gfCNCPoint1[22811] = {X 129.1532, Y 40.1052, Z -2.1667, A 0.000, B 0.000, C 0.000 }
gfCNCPoint1[22812] = {X 131.4548, Y 40.7854, Z -2.1667, A 0.000, B 0.000, C 0.000 }
gfCNCPoint1[22813] = {X 131.9017, Y 39.5320, Z -2.1667, A 0.000, B 0.000, C 0.000 }
gfCNCPoint1[22814] = {X 132.4836, Y 38.3354, Z -2.1667, A 0.000, B 0.000, C 0.000 }
gfCNCPoint1[22815] = {X 132.4836, Y 29.5202, Z -2.1667, A 0.000, B 0.000, C 0.000 }
gfCNCPoint1[22816] = {X 131.3523, Y 29.3993, Z -2.1667, A 0.000, B 0.000, C 0.000 }
gfCNCPoint1[22817] = {X 130.2373, Y 29.1724, Z -2.1667, A 0.000, B 0.000, C 0.000 }
gfCNCPoint1[22818] = {X 129.1487, Y 28.8417, Z -2.1667, A 0.000, B 0.000, C 0.000 }
gfCNCPoint1[22819] = {X 128.0242, Y 28.3763, Z -2.1667, A 0.000, B 0.000, C 0.000 }
gfCNCPoint1[22820] = {X 126.9523, Y 27.8001, Z -2.1667, A 0.000, B 0.000, C 0.000 }
gfCNCPoint1[22821] = {X 125.9438, Y 27.1189, Z -2.1667, A 0.000, B 0.000, C 0.000 }
gfCNCPoint1[22822] = {X 125.9432, Y 38.9884, Z -2.1667, A 0.000, B 0.000, C 0.000 }
gfCNCPoint1[22823] = {X 126.4735, Y 39.9279, Z -2.1667, A 0.000, B 0.000, C 0.000 }
gfCNCPoint1[22824] = {X 126.8960, Y 40.9205, Z -2.1667, A 0.000, B 0.000, C 0.000 }
gfCNCPoint1[22825] = {X 127.2098, Y 41.9730, Z -2.1667, A 0.000, B 0.000, C 0.000 }
gfCNCPoint1[22826] = {X 127.4025, Y 43.0542, Z -2.1667, A 0.000, B 0.000, C 0.000 }
gfCNCPoint1[22827] = {X 127.4714, Y 44.1502, Z -2.1667, A 0.000, B 0.000, C 0.000 }
gfCNCPoint1[22828] = {X 127.4716, Y 45.0000, Z -2.1667, A 0.000, B 0.000, C 0.000 }
gfCNCPoint1[22829] = {X 127.4070, Y 46.1159, Z -2.1667, A 0.000, B 0.000, C 0.000 }
gfCNCPoint1[22830] = {X 127.2143, Y 47.2168, Z -2.1667, A 0.000, B 0.000, C 0.000 }
gfCNCPoint1[22831] = {X 126.8960, Y 48.2883, Z -2.1667, A 0.000, B 0.000, C 0.000 }
gfCNCPoint1[22832] = {X 126.2883, Y 49.6376, Z -2.1667, A 0.000, B 0.000, C 0.000 }
gfCNCPoint1[22833] = {X 125.4821, Y 50.8786, Z -2.1667, A 0.000, B 0.000, C 0.000 }
gfCNCPoint1[22834] = {X 124.4962, Y 51.9821, Z -2.1667, A 0.000, B 0.000, C 0.000 }
gfCNCPoint1[22835] = {X 123.3536, Y 52.9225, Z -2.1667, A 0.000, B 0.000, C 0.000 }
gfCNCPoint1[22836] = {X 122.0810, Y 53.6778, Z -2.1667, A 0.000, B 0.000, C 0.000 }
gfCNCPoint1[22837] = {X 120.7081, Y 54.2302, Z -2.1667, A 0.000, B 0.000, C 0.000 }
gfCNCPoint1[22838] = {X 119.2671, Y 54.5669, Z -2.1667, A 0.000, B 0.000, C 0.000 }
gfCNCPoint1[22839] = {X 117.7916, Y 54.6800, Z -2.1667, A 0.000, B 0.000, C 0.000 }
gfCNCPoint1[22840] = {X 111.9185, Y 54.6800, Z -2.1667, A 0.000, B 0.000, C 0.000 }
gfCNCPoint1[22841] = {X 110.6386, Y 54.5950, Z -2.1667, A 0.000, B 0.000, C 0.000 }
gfCNCPoint1[22842] = {X 109.3812, Y 54.3415, Z -2.1667, A 0.000, B 0.000, C 0.000 }
gfCNCPoint1[22843] = {X 108.1683, Y 53.9240, Z -2.1667, A 0.000, B 0.000, C 0.000 }
gfCNCPoint1[22844] = {X 107.0213, Y 53.3498, Z -2.1667, A 0.000, B 0.000, C 0.000 }
gfCNCPoint1[22845] = {X 106.6480, Y 53.5578, Z -2.1667, A 0.000, B 0.000, C 0.000 }
gfCNCPoint1[22846] = {X 106.2658, Y 53.7492, Z -2.1667, A 0.000, B 0.000, C 0.000 }
gfCNCPoint1[22847] = {X 105.0149, Y 54.2382, Z -2.1667, A 0.000, B 0.000, C 0.000 }
gfCNCPoint1[22848] = {X 103.7084, Y 54.5495, Z -2.1667, A 0.000, B 0.000, C 0.000 }
gfCNCPoint1[22849] = {X 102.3713, Y 54.6768, Z -2.1667, A 0.000, B 0.000, C 0.000 }
gfCNCPoint1[22850] = {X 101.0295, Y 54.6179, Z -2.1667, A 0.000, B 0.000, C 0.000 }
gfCNCPoint1[22851] = {X 99.7088, Y 54.3738, Z -2.1667, A 0.000, B 0.000, C 0.000 }
gfCNCPoint1[22852] = {X 98.4345, Y 53.9493, Z -2.1667, A 0.000, B 0.000, C 0.000 }
gfCNCPoint1[22853] = {X 97.2313, Y 53.3524, Z -2.1667, A 0.000, B 0.000, C 0.000 }
gfCNCPoint1[22854] = {X 96.0852, Y 53.9255, Z -2.1667, A 0.000, B 0.000, C 0.000 }
gfCNCPoint1[22855] = {X 94.8734, Y 54.3422, Z -2.1667, A 0.000, B 0.000, C 0.000 }
gfCNCPoint1[22856] = {X 93.6172, Y 54.5952, Z -2.1667, A 0.000, B 0.000, C 0.000 }
gfCNCPoint1[22857] = {X 92.3385, Y 54.6800, Z -2.1667, A 0.000, B 0.000, C 0.000 }
gfCNCPoint1[22858] = {X 85.8951, Y 54.6800, Z -2.1667, A 0.000, B 0.000, C 0.000 }
gfCNCPoint1[22859] = {X 84.6159, Y 54.5951, Z -2.1667, A 0.000, B 0.000, C 0.000 }
gfCNCPoint1[22860] = {X 83.3592, Y 54.3419, Z -2.1667, A 0.000, B 0.000, C 0.000 }
gfCNCPoint1[22861] = {X 82.1469, Y 53.9249, Z -2.1667, A 0.000, B 0.000, C 0.000 }
gfCNCPoint1[22862] = {X 81.0644, Y 55.1572, Z -2.1667, A 0.000, B 0.000, C 0.000 }
gfCNCPoint1[22863] = {X 79.8495, Y 56.2591, Z -2.1667, A 0.000, B 0.000, C 0.000 }
gfCNCPoint1[22864] = {X 78.5178, Y 57.2166, Z -2.1667, A 0.000, B 0.000, C 0.000 }
gfCNCPoint1[22865] = {X 77.0863, Y 58.0174, Z -2.1667, A 0.000, B 0.000, C 0.000 }
gfCNCPoint1[22866] = {X 75.5734, Y 58.6511, Z -2.1667, A 0.000, B 0.000, C 0.000 }
gfCNCPoint1[22867] = {X 73.9986, Y 59.1096, Z -2.1667, A 0.000, B 0.000, C 0.000 }
gfCNCPoint1[22868] = {X 72.3820, Y 59.3871, Z -2.1667, A 0.000, B 0.000, C 0.000 }
gfCNCPoint1[22869] = {X 70.7445, Y 59.4800, Z -2.1667, A 0.000, B 0.000, C 0.000 }
gfCNCPoint1[22870] = {X 64.1851, Y 59.4800, Z -2.1667, A 0.000, B 0.000, C 0.000 }
gfCNCPoint1[22871] = {X 62.4203, Y 59.3720, Z -2.1667, A 0.000, B 0.000, C 0.000 }
gfCNCPoint1[22872] = {X 60.6818, Y 59.0498, Z -2.1667, A 0.000, B 0.000, C 0.000 }
gfCNCPoint1[22873] = {X 58.9955, Y 58.5181, Z -2.1667, A 0.000, B 0.000, C 0.000 }
gfCNCPoint1[22874] = {X 57.3866, Y 57.7848, Z -2.1667, A 0.000, B 0.000, C 0.000 }
gfCNCPoint1[22875] = {X 55.8790, Y 56.8608, Z -2.1667, A 0.000, B 0.000, C 0.000 }
gfCNCPoint1[22876] = {X 54.3715, Y 57.7848, Z -2.1667, A 0.000, B 0.000, C 0.000 }
gfCNCPoint1[22877] = {X 52.7626, Y 58.5181, Z -2.1667, A 0.000, B 0.000, C 0.000 }
gfCNCPoint1[22878] = {X 51.0763, Y 59.0498, Z -2.1667, A 0.000, B 0.000, C 0.000 }
gfCNCPoint1[22879] = {X 49.3378, Y 59.3720, Z -2.1667, A 0.000, B 0.000, C 0.000 }
gfCNCPoint1[22880] = {X 47.5729, Y 59.4800, Z -2.1667, A 0.000, B 0.000, C 0.000 }
gfCNCPoint1[22881] = {X 40.6393, Y 59.4800, Z -2.1667, A 0.000, B 0.000, C 0.000 }
gfCNCPoint1[22882] = {X 38.9795, Y 59.3845, Z -2.1667, A 0.000, B 0.000, C 0.000 }
gfCNCPoint1[22883] = {X 37.3415, Y 59.0995, Z -2.1667, A 0.000, B 0.000, C 0.000 }
gfCNCPoint1[22884] = {X 35.7470, Y 58.6285, Z -2.1667, A 0.000, B 0.000, C 0.000 }
gfCNCPoint1[22885] = {X 34.0331, Y 59.4863, Z -2.1667, A 0.000, B 0.000, C 0.000 }
gfCNCPoint1[22886] = {X 32.2408, Y 60.1653, Z -2.1667, A 0.000, B 0.000, C 0.000 }
gfCNCPoint1[22887] = {X 30.3888, Y 60.6585, Z -2.1667, A 0.000, B 0.000, C 0.000 }
gfCNCPoint1[22888] = {X 28.4962, Y 60.9608, Z -2.1667, A 0.000, B 0.000, C 0.000 }
gfCNCPoint1[22889] = {X 25.7981, Y 62.0563, Z -2.1667, A 0.000, B 0.000, C 0.000 }
gfCNCPoint1[22890] = {X 23.0321, Y 62.9667, Z -2.1667, A 0.000, B 0.000, C 0.000 }
gfCNCPoint1[22891] = {X 20.1653, Y 63.6947, Z -2.1667, A 0.000, B 0.000, C 0.000 }
gfCNCPoint1[22892] = {X 17.2496, Y 64.1921, Z -2.1667, A 0.000, B 0.000, C 0.000 }
gfCNCPoint1[22893] = {X 14.3035, Y 64.4558, Z -2.1667, A 0.000, B 0.000, C 0.000 }
gfCNCPoint1[22894] = {X 14.3035, Y 85.6949, Z -2.1667, A 0.000, B 0.000, C 0.000 }
gfCNCPoint1[22895] = {X 112.5246, Y 85.6949, Z -2.1667, A 0.000, B 0.000, C 0.000 }
gfCNCPoint1[22896] = {X 113.6274, Y 84.5920, Z -2.1667, A 0.000, B 0.000, C 0.000 }
gfCNCPoint1[22897] = {X 114.8273, Y 83.5956, Z -2.1667, A 0.000, B 0.000, C 0.000 }
gfCNCPoint1[22898] = {X 116.1140, Y 82.7142, Z -2.1667, A 0.000, B 0.000, C 0.000 }
gfCNCPoint1[22899] = {X 117.4766, Y 81.9553, Z -2.1667, A 0.000, B 0.000, C 0.000 }
gfCNCPoint1[22900] = {X 111.0585, Y 69.0646, Z -2.1667, A 0.000, B 0.000, C 0.000 }
gfCNCPoint1[22901] = {X 109.0296, Y 68.9061, Z -2.1667, A 0.000, B 0.000, C 0.000 }
gfCNCPoint1[22902] = {X 107.0213, Y 68.5768, Z -2.1667, A 0.000, B 0.000, C 0.000 }
gfCNCPoint1[22903] = {X 105.0765, Y 68.8983, Z -2.1667, A 0.000, B 0.000, C 0.000 }
gfCNCPoint1[22904] = {X 103.1119, Y 69.0597, Z -2.1667, A 0.000, B 0.000, C 0.000 }
gfCNCPoint1[22905] = {X 101.1407, Y 69.0599, Z -2.1667, A 0.000, B 0.000, C 0.000 }
gfCNCPoint1[22906] = {X 99.1761, Y 68.8989, Z -2.1667, A 0.000, B 0.000, C 0.000 }
gfCNCPoint1[22907] = {X 97.2313, Y 68.5777, Z -2.1667, A 0.000, B 0.000, C 0.000 }
gfCNCPoint1[22908] = {X 95.6131, Y 68.8563, Z -2.1667, A 0.000, B 0.000, C 0.000 }
gfCNCPoint1[22909] = {X 93.9796, Y 69.0240, Z -2.1667, A 0.000, B 0.000, C 0.000 }
gfCNCPoint1[22910] = {X 92.3385, Y 69.0800, Z -2.1667, A 0.000, B 0.000, C 0.000 }
gfCNCPoint1[22911] = {X 86.6884, Y 69.0800, Z -2.1667, A 0.000, B 0.000, C 0.000 }
gfCNCPoint1[22912] = {X 84.7317, Y 70.2668, Z -2.1667, A 0.000, B 0.000, C 0.000 }
gfCNCPoint1[22913] = {X 82.6873, Y 71.2949, Z -2.1667, A 0.000, B 0.000, C 0.000 }
gfCNCPoint1[22914] = {X 107.2717, Y 71.2949, Z -2.1667, A 0.000, B 0.000, C 0.000 }
gfCNCPoint1[22915] = {X 109.1259, Y 70.1132, Z -2.1667, A 0.000, B 0.000, C 0.000 }
gfCNCPoint1[22916] = {X 111.0585, Y 69.0646, Z -2.1667, A 0.000, B 0.000, C 0.000 }
gfCNCPoint1[22917] = {X 112.1282, Y 71.2131, Z -2.1667, A 0.000, B 0.000, C 0.000 }
gfCNCPoint1[22918] = {X 113.1274, Y 70.7392, Z -2.1667, A 0.000, B 0.000, C 0.000 }
gfCNCPoint1[22919] = {X 114.1439, Y 70.3040, Z -2.1667, A 0.000, B 0.000, C 0.000 }
gfCNCPoint1[22920] = {X 117.4441, Y 66.6800, Z -2.1667, A 0.000, B 0.000, C 0.000 }
gfCNCPoint1[22921] = {X 111.9185, Y 66.6800, Z -2.1667, A 0.000, B 0.000, C 0.000 }
gfCNCPoint1[22922] = {X 111.5313, Y 66.6765, Z -2.1667, A 0.000, B 0.000, C 0.000 }
gfCNCPoint1[22923] = {X 111.1442, Y 66.6662, Z -2.1667, A 0.000, B 0.000, C 0.000 }
gfCNCPoint1[22924] = {X 109.0696, Y 66.4920, Z -2.1667, A 0.000, B 0.000, C 0.000 }
gfCNCPoint1[22925] = {X 107.0213, Y 66.1197, Z -2.1667, A 0.000, B 0.000, C 0.000 }
gfCNCPoint1[22926] = {X 105.0796, Y 66.4776, Z -2.1667, A 0.000, B 0.000, C 0.000 }
gfCNCPoint1[22927] = {X 103.1135, Y 66.6574, Z -2.1667, A 0.000, B 0.000, C 0.000 }
gfCNCPoint1[22928] = {X 101.1392, Y 66.6576, Z -2.1667, A 0.000, B 0.000, C 0.000 }
gfCNCPoint1[22929] = {X 99.1730, Y 66.4782, Z -2.1667, A 0.000, B 0.000, C 0.000 }
gfCNCPoint1[22930] = {X 97.2313, Y 66.1207, Z -2.1667, A 0.000, B 0.000, C 0.000 }
gfCNCPoint1[22931] = {X 95.6161, Y 66.4308, Z -2.1667, A 0.000, B 0.000, C 0.000 }
gfCNCPoint1[22932] = {X 93.9821, Y 66.6176, Z -2.1667, A 0.000, B 0.000, C 0.000 }
gfCNCPoint1[22933] = {X 92.3385, Y 66.6800, Z -2.1667, A 0.000, B 0.000, C 0.000 }
gfCNCPoint1[22934] = {X 85.9487, Y 66.6800, Z -2.1667, A 0.000, B 0.000, C 0.000 }
gfCNCPoint1[22935] = {X 83.8781, Y 67.9935, Z -2.1667, A 0.000, B 0.000, C 0.000 }
gfCNCPoint1[22936] = {X 81.6948, Y 69.1097, Z -2.1667, A 0.000, B 0.000, C 0.000 }
gfCNCPoint1[22937] = {X 79.6018, Y 69.9547, Z -2.1667, A 0.000, B 0.000, C 0.000 }
gfCNCPoint1[22938] = {X 77.4444, Y 70.6184, Z -2.1667, A 0.000, B 0.000, C 0.000 }
gfCNCPoint1[22939] = {X 75.2383, Y 71.0959, Z -2.1667, A 0.000, B 0.000, C 0.000 }
gfCNCPoint1[22940] = {X 72.9996, Y 71.3838, Z -2.1667, A 0.000, B 0.000, C 0.000 }
gfCNCPoint1[22941] = {X 70.7445, Y 71.4800, Z -2.1667, A 0.000, B 0.000, C 0.000 }
gfCNCPoint1[22942] = {X 64.1851, Y 71.4800, Z -2.1667, A 0.000, B 0.000, C 0.000 }
gfCNCPoint1[22943] = {X 62.0752, Y 71.3958, Z -2.1667, A 0.000, B 0.000, C 0.000 }
gfCNCPoint1[22944] = {X 59.9787, Y 71.1438, Z -2.1667, A 0.000, B 0.000, C 0.000 }
gfCNCPoint1[22945] = {X 57.9089, Y 70.7255, Z -2.1667, A 0.000, B 0.000, C 0.000 }
gfCNCPoint1[22946] = {X 55.8790, Y 70.1436, Z -2.1667, A 0.000, B 0.000, C 0.000 }
gfCNCPoint1[22947] = {X 53.8492, Y 70.7255, Z -2.1667, A 0.000, B 0.000, C 0.000 }
gfCNCPoint1[22948] = {X 51.7794, Y 71.1438, Z -2.1667, A 0.000, B 0.000, C 0.000 }
gfCNCPoint1[22949] = {X 49.6829, Y 71.3958, Z -2.1667, A 0.000, B 0.000, C 0.000 }
gfCNCPoint1[22950] = {X 47.5729, Y 71.4800, Z -2.1667, A 0.000, B 0.000, C 0.000 }
gfCNCPoint1[22951] = {X 40.6393, Y 71.4800, Z -2.1667, A 0.000, B 0.000, C 0.000 }
gfCNCPoint1[22952] = {X 38.8042, Y 71.4163, Z -2.1667, A 0.000, B 0.000, C 0.000 }
gfCNCPoint1[22953] = {X 36.9779, Y 71.2256, Z -2.1667, A 0.000, B 0.000, C 0.000 }
gfCNCPoint1[22954] = {X 34.3998, Y 72.0339, Z -2.1667, A 0.000, B 0.000, C 0.000 }
gfCNCPoint1[22955] = {X 31.7610, Y 72.6132, Z -2.1667, A 0.000, B 0.000, C 0.000 }
gfCNCPoint1[22956] = {X 30.3294, Y 73.1742, Z -2.1667, A 0.000, B 0.000, C 0.000 }
gfCNCPoint1[22957] = {X 28.8828, Y 73.6949, Z -2.1667, A 0.000, B 0.000, C 0.000 }
gfCNCPoint1[22958] = {X 108.0339, Y 73.6949, Z -2.1667, A 0.000, B 0.000, C 0.000 }
gfCNCPoint1[22959] = {X 110.0295, Y 72.3690, Z -2.1667, A 0.000, B 0.000, C 0.000 }
gfCNCPoint1[22960] = {X 112.1282, Y 71.2131, Z -2.1667, A 0.000, B 0.000, C 0.000 }
gfCNCPoint1[22961] = {X 113.1979, Y 73.3615, Z -2.1667, A 0.000, B 0.000, C 0.000 }
gfCNCPoint1[22962] = {X 114.3580, Y 72.8185, Z -2.1667, A 0.000, B 0.000, C 0.000 }
gfCNCPoint1[22963] = {X 115.5430, Y 72.3323, Z -2.1667, A 0.000, B 0.000, C 0.000 }
gfCNCPoint1[22964] = {X 123.7288, Y 63.3431, Z -2.1667, A 0.000, B 0.000, C 0.000 }
gfCNCPoint1[22965] = {X 121.7860, Y 63.8617, Z -2.1667, A 0.000, B 0.000, C 0.000 }
gfCNCPoint1[22966] = {X 119.7997, Y 64.1751, Z -2.1667, A 0.000, B 0.000, C 0.000 }
gfCNCPoint1[22967] = {X 117.7916, Y 64.2800, Z -2.1667, A 0.000, B 0.000, C 0.000 }
gfCNCPoint1[22968] = {X 111.9185, Y 64.2800, Z -2.1667, A 0.000, B 0.000, C 0.000 }
gfCNCPoint1[22969] = {X 110.2700, Y 64.2094, Z -2.1667, A 0.000, B 0.000, C 0.000 }
gfCNCPoint1[22970] = {X 108.6336, Y 63.9981, Z -2.1667, A 0.000, B 0.000, C 0.000 }
gfCNCPoint1[22971] = {X 107.0213, Y 63.6477, Z -2.1667, A 0.000, B 0.000, C 0.000 }
gfCNCPoint1[22972] = {X 105.0841, Y 64.0514, Z -2.1667, A 0.000, B 0.000, C 0.000 }
gfCNCPoint1[22973] = {X 103.1158, Y 64.2545, Z -2.1667, A 0.000, B 0.000, C 0.000 }
gfCNCPoint1[22974] = {X 101.1370, Y 64.2547, Z -2.1667, A 0.000, B 0.000, C 0.000 }
gfCNCPoint1[22975] = {X 99.1686, Y 64.0521, Z -2.1667, A 0.000, B 0.000, C 0.000 }
gfCNCPoint1[22976] = {X 97.2313, Y 63.6488, Z -2.1667, A 0.000, B 0.000, C 0.000 }
gfCNCPoint1[22977] = {X 95.6204, Y 63.9986, Z -2.1667, A 0.000, B 0.000, C 0.000 }
gfCNCPoint1[22978] = {X 93.9855, Y 64.2095, Z -2.1667, A 0.000, B 0.000, C 0.000 }
gfCNCPoint1[22979] = {X 92.3385, Y 64.2800, Z -2.1667, A 0.000, B 0.000, C 0.000 }
gfCNCPoint1[22980] = {X 85.8951, Y 64.2800, Z -2.1667, A 0.000, B 0.000, C 0.000 }
gfCNCPoint1[22981] = {X 85.5417, Y 64.2768, Z -2.1667, A 0.000, B 0.000, C 0.000 }
gfCNCPoint1[22982] = {X 85.1884, Y 64.2670, Z -2.1667, A 0.000, B 0.000, C 0.000 }
gfCNCPoint1[22983] = {X 83.3593, Y 65.5113, Z -2.1667, A 0.000, B 0.000, C 0.000 }
gfCNCPoint1[22984] = {X 81.4238, Y 66.5824, Z -2.1667, A 0.000, B 0.000, C 0.000 }
gfCNCPoint1[22985] = {X 79.3981, Y 67.4713, Z -2.1667, A 0.000, B 0.000, C 0.000 }
gfCNCPoint1[22986] = {X 77.2994, Y 68.1706, Z -2.1667, A 0.000, B 0.000, C 0.000 }
gfCNCPoint1[22987] = {X 75.1454, Y 68.6744, Z -2.1667, A 0.000, B 0.000, C 0.000 }
gfCNCPoint1[22988] = {X 72.9543, Y 68.9784, Z -2.1667, A 0.000, B 0.000, C 0.000 }
gfCNCPoint1[22989] = {X 70.7445, Y 69.0800, Z -2.1667, A 0.000, B 0.000, C 0.000 }
gfCNCPoint1[22990] = {X 64.1851, Y 69.0800, Z -2.1667, A 0.000, B 0.000, C 0.000 }
gfCNCPoint1[22991] = {X 62.0678, Y 68.9867, Z -2.1667, A 0.000, B 0.000, C 0.000 }
gfCNCPoint1[22992] = {X 59.9669, Y 68.7076, Z -2.1667, A 0.000, B 0.000, C 0.000 }
gfCNCPoint1[22993] = {X 57.8986, Y 68.2449, Z -2.1667, A 0.000, B 0.000, C 0.000 }
gfCNCPoint1[22994] = {X 55.8790, Y 67.6021, Z -2.1667, A 0.000, B 0.000, C 0.000 }
gfCNCPoint1[22995] = {X 53.8595, Y 68.2449, Z -2.1667, A 0.000, B 0.000, C 0.000 }
gfCNCPoint1[22996] = {X 51.7912, Y 68.7076, Z -2.1667, A 0.000, B 0.000, C 0.000 }
gfCNCPoint1[22997] = {X 49.6903, Y 68.9867, Z -2.1667, A 0.000, B 0.000, C 0.000 }
gfCNCPoint1[22998] = {X 47.5729, Y 69.0800, Z -2.1667, A 0.000, B 0.000, C 0.000 }
gfCNCPoint1[22999] = {X 40.6393, Y 69.0800, Z -2.1667, A 0.000, B 0.000, C 0.000 }
gfCNCPoint1[23000] = {X 38.6738, Y 68.9996, Z -2.1667, A 0.000, B 0.000, C 0.000 }
gfCNCPoint1[23001] = {X 36.7214, Y 68.7591, Z -2.1667, A 0.000, B 0.000, C 0.000 }
gfCNCPoint1[23002] = {X 34.8828, Y 69.3981, Z -2.1667, A 0.000, B 0.000, C 0.000 }
gfCNCPoint1[23003] = {X 33.0048, Y 69.9097, Z -2.1667, A 0.000, B 0.000, C 0.000 }
gfCNCPoint1[23004] = {X 31.0962, Y 70.2916, Z -2.1667, A 0.000, B 0.000, C 0.000 }
gfCNCPoint1[23005] = {X 29.6075, Y 70.8814, Z -2.1667, A 0.000, B 0.000, C 0.000 }
gfCNCPoint1[23006] = {X 28.1016, Y 71.4256, Z -2.1667, A 0.000, B 0.000, C 0.000 }
gfCNCPoint1[23007] = {X 26.9268, Y 71.8147, Z -2.1667, A 0.000, B 0.000, C 0.000 }
gfCNCPoint1[23008] = {X 25.7433, Y 72.1759, Z -2.1667, A 0.000, B 0.000, C 0.000 }
gfCNCPoint1[23009] = {X 24.8260, Y 72.4376, Z -2.1667, A 0.000, B 0.000, C 0.000 }
gfCNCPoint1[23010] = {X 23.9035, Y 72.6805, Z -2.1667, A 0.000, B 0.000, C 0.000 }
gfCNCPoint1[23011] = {X 23.9035, Y 76.0949, Z -2.1667, A 0.000, B 0.000, C 0.000 }
gfCNCPoint1[23012] = {X 108.8319, Y 76.0949, Z -2.1667, A 0.000, B 0.000, C 0.000 }
gfCNCPoint1[23013] = {X 110.2270, Y 75.0898, Z -2.1667, A 0.000, B 0.000, C 0.000 }
gfCNCPoint1[23014] = {X 111.6843, Y 74.1774, Z -2.1667, A 0.000, B 0.000, C 0.000 }
gfCNCPoint1[23015] = {X 113.1979, Y 73.3615, Z -2.1667, A 0.000, B 0.000, C 0.000 }
gfCNCPoint1[23016] = {X 114.2675, Y 75.5099, Z -2.1667, A 0.000, B 0.000, C 0.000 }
gfCNCPoint1[23017] = {X 115.5786, Y 74.9055, Z -2.1667, A 0.000, B 0.000, C 0.000 }
gfCNCPoint1[23018] = {X 116.9235, Y 74.3808, Z -2.1667, A 0.000, B 0.000, C 0.000 }
gfCNCPoint1[23019] = {X 130.4117, Y 59.5689, Z -2.1667, A 0.000, B 0.000, C 0.000 }
gfCNCPoint1[23020] = {X 129.5280, Y 58.7534, Z -2.1667, A 0.000, B 0.000, C 0.000 }
gfCNCPoint1[23021] = {X 128.6970, Y 57.8844, Z -2.1667, A 0.000, B 0.000, C 0.000 }
gfCNCPoint1[23022] = {X 127.3931, Y 58.8832, Z -2.1667, A 0.000, B 0.000, C 0.000 }
gfCNCPoint1[23023] = {X 125.9984, Y 59.7507, Z -2.1667, A 0.000, B 0.000, C 0.000 }
gfCNCPoint1[23024] = {X 124.5259, Y 60.4785, Z -2.1667, A 0.000, B 0.000, C 0.000 }
gfCNCPoint1[23025] = {X 122.9897, Y 61.0597, Z -2.1667, A 0.000, B 0.000, C 0.000 }
gfCNCPoint1[23026] = {X 121.2887, Y 61.5138, Z -2.1667, A 0.000, B 0.000, C 0.000 }
gfCNCPoint1[23027] = {X 119.5497, Y 61.7882, Z -2.1667, A 0.000, B 0.000, C 0.000 }
gfCNCPoint1[23028] = {X 117.7916, Y 61.8800, Z -2.1667, A 0.000, B 0.000, C 0.000 }
gfCNCPoint1[23029] = {X 111.9185, Y 61.8800, Z -2.1667, A 0.000, B 0.000, C 0.000 }
gfCNCPoint1[23030] = {X 110.2649, Y 61.7988, Z -2.1667, A 0.000, B 0.000, C 0.000 }
gfCNCPoint1[23031] = {X 108.6273, Y 61.5560, Z -2.1667, A 0.000, B 0.000, C 0.000 }
gfCNCPoint1[23032] = {X 107.0213, Y 61.1540, Z -2.1667, A 0.000, B 0.000, C 0.000 }
gfCNCPoint1[23033] = {X 105.0907, Y 61.6173, Z -2.1667, A 0.000, B 0.000, C 0.000 }
gfCNCPoint1[23034] = {X 103.1191, Y 61.8506, Z -2.1667, A 0.000, B 0.000, C 0.000 }
gfCNCPoint1[23035] = {X 101.1337, Y 61.8509, Z -2.1667, A 0.000, B 0.000, C 0.000 }
gfCNCPoint1[23036] = {X 99.1620, Y 61.6181, Z -2.1667, A 0.000, B 0.000, C 0.000 }
gfCNCPoint1[23037] = {X 97.2313, Y 61.1553, Z -2.1667, A 0.000, B 0.000, C 0.000 }
gfCNCPoint1[23038] = {X 95.6267, Y 61.5566, Z -2.1667, A 0.000, B 0.000, C 0.000 }
gfCNCPoint1[23039] = {X 93.9906, Y 61.7990, Z -2.1667, A 0.000, B 0.000, C 0.000 }
gfCNCPoint1[23040] = {X 92.3385, Y 61.8800, Z -2.1667, A 0.000, B 0.000, C 0.000 }
gfCNCPoint1[23041] = {X 85.8951, Y 61.8800, Z -2.1667, A 0.000, B 0.000, C 0.000 }
gfCNCPoint1[23042] = {X 85.1609, Y 61.8640, Z -2.1667, A 0.000, B 0.000, C 0.000 }
gfCNCPoint1[23043] = {X 84.4280, Y 61.8161, Z -2.1667, A 0.000, B 0.000, C 0.000 }
gfCNCPoint1[23044] = {X 82.7246, Y 63.0692, Z -2.1667, A 0.000, B 0.000, C 0.000 }
gfCNCPoint1[23045] = {X 80.9073, Y 64.1504, Z -2.1667, A 0.000, B 0.000, C 0.000 }
gfCNCPoint1[23046] = {X 78.9932, Y 65.0494, Z -2.1667, A 0.000, B 0.000, C 0.000 }
gfCNCPoint1[23047] = {X 77.0007, Y 65.7577, Z -2.1667, A 0.000, B 0.000, C 0.000 }
gfCNCPoint1[23048] = {X 74.9487, Y 66.2685, Z -2.1667, A 0.000, B 0.000, C 0.000 }
gfCNCPoint1[23049] = {X 72.8566, Y 66.5769, Z -2.1667, A 0.000, B 0.000, C 0.000 }
gfCNCPoint1[23050] = {X 70.7445, Y 66.6800, Z -2.1667, A 0.000, B 0.000, C 0.000 }
gfCNCPoint1[23051] = {X 64.1851, Y 66.6800, Z -2.1667, A 0.000, B 0.000, C 0.000 }
gfCNCPoint1[23052] = {X 62.0576, Y 66.5753, Z -2.1667, A 0.000, B 0.000, C 0.000 }
gfCNCPoint1[23053] = {X 59.9505, Y 66.2624, Z -2.1667, A 0.000, B 0.000, C 0.000 }
gfCNCPoint1[23054] = {X 57.8844, Y 65.7442, Z -2.1667, A 0.000, B 0.000, C 0.000 }
gfCNCPoint1[23055] = {X 55.8790, Y 65.0258, Z -2.1667, A 0.000, B 0.000, C 0.000 }
gfCNCPoint1[23056] = {X 53.8737, Y 65.7442, Z -2.1667, A 0.000, B 0.000, C 0.000 }
gfCNCPoint1[23057] = {X 51.8075, Y 66.2624, Z -2.1667, A 0.000, B 0.000, C 0.000 }
gfCNCPoint1[23058] = {X 49.7005, Y 66.5753, Z -2.1667, A 0.000, B 0.000, C 0.000 }
gfCNCPoint1[23059] = {X 47.5729, Y 66.6800, Z -2.1667, A 0.000, B 0.000, C 0.000 }
gfCNCPoint1[23060] = {X 40.6393, Y 66.6800, Z -2.1667, A 0.000, B 0.000, C 0.000 }
gfCNCPoint1[23061] = {X 38.5440, Y 66.5785, Z -2.1667, A 0.000, B 0.000, C 0.000 }
gfCNCPoint1[23062] = {X 36.4684, Y 66.2750, Z -2.1667, A 0.000, B 0.000, C 0.000 }
gfCNCPoint1[23063] = {X 34.5052, Y 67.0002, Z -2.1667, A 0.000, B 0.000, C 0.000 }
gfCNCPoint1[23064] = {X 32.4901, Y 67.5653, Z -2.1667, A 0.000, B 0.000, C 0.000 }
gfCNCPoint1[23065] = {X 30.4361, Y 67.9665, Z -2.1667, A 0.000, B 0.000, C 0.000 }
gfCNCPoint1[23066] = {X 27.7779, Y 68.9963, Z -2.1667, A 0.000, B 0.000, C 0.000 }
gfCNCPoint1[23067] = {X 25.0655, Y 69.8736, Z -2.1667, A 0.000, B 0.000, C 0.000 }
gfCNCPoint1[23068] = {X 23.2938, Y 70.3591, Z -2.1667, A 0.000, B 0.000, C 0.000 }
gfCNCPoint1[23069] = {X 21.5035, Y 70.7708, Z -2.1667, A 0.000, B 0.000, C 0.000 }
gfCNCPoint1[23070] = {X 21.5035, Y 78.4949, Z -2.1667, A 0.000, B 0.000, C 0.000 }
gfCNCPoint1[23071] = {X 109.6715, Y 78.4949, Z -2.1667, A 0.000, B 0.000, C 0.000 }
gfCNCPoint1[23072] = {X 111.1263, Y 77.3843, Z -2.1667, A 0.000, B 0.000, C 0.000 }
gfCNCPoint1[23073] = {X 112.6613, Y 76.3874, Z -2.1667, A 0.000, B 0.000, C 0.000 }
gfCNCPoint1[23074] = {X 114.2675, Y 75.5099, Z -2.1667, A 0.000, B 0.000, C 0.000 }
gfCNCPoint1[23075] = {X 115.3372, Y 77.6584, Z -2.1667, A 0.000, B 0.000, C 0.000 }
gfCNCPoint1[23076] = {X 116.7878, Y 77.0015, Z -2.1667, A 0.000, B 0.000, C 0.000 }
gfCNCPoint1[23077] = {X 118.2826, Y 76.4529, Z -2.1667, A 0.000, B 0.000, C 0.000 }
gfCNCPoint1[23078] = {X 133.9639, Y 59.2326, Z -2.1667, A 0.000, B 0.000, C 0.000 }
gfCNCPoint1[23079] = {X 132.7159, Y 58.3550, Z -2.1667, A 0.000, B 0.000, C 0.000 }
gfCNCPoint1[23080] = {X 131.5522, Y 57.3683, Z -2.1667, A 0.000, B 0.000, C 0.000 }
gfCNCPoint1[23081] = {X 130.4824, Y 56.2805, Z -2.1667, A 0.000, B 0.000, C 0.000 }
gfCNCPoint1[23082] = {X 129.6655, Y 55.2988, Z -2.1667, A 0.000, B 0.000, C 0.000 }
gfCNCPoint1[23083] = {X 128.9251, Y 54.2582, Z -2.1667, A 0.000, B 0.000, C 0.000 }
gfCNCPoint1[23084] = {X 128.0750, Y 55.1942, Z -2.1667, A 0.000, B 0.000, C 0.000 }
gfCNCPoint1[23085] = {X 127.1464, Y 56.0525, Z -2.1667, A 0.000, B 0.000, C 0.000 }
gfCNCPoint1[23086] = {X 125.7915, Y 57.0695, Z -2.1667, A 0.000, B 0.000, C 0.000 }
gfCNCPoint1[23087] = {X 124.3270, Y 57.9212, Z -2.1667, A 0.000, B 0.000, C 0.000 }
gfCNCPoint1[23088] = {X 122.7731, Y 58.5961, Z -2.1667, A 0.000, B 0.000, C 0.000 }
gfCNCPoint1[23089] = {X 121.1510, Y 59.0849, Z -2.1667, A 0.000, B 0.000, C 0.000 }
gfCNCPoint1[23090] = {X 119.4828, Y 59.3809, Z -2.1667, A 0.000, B 0.000, C 0.000 }
gfCNCPoint1[23091] = {X 117.7916, Y 59.4800, Z -2.1667, A 0.000, B 0.000, C 0.000 }
gfCNCPoint1[23092] = {X 111.9185, Y 59.4800, Z -2.1667, A 0.000, B 0.000, C 0.000 }
gfCNCPoint1[23093] = {X 110.2569, Y 59.3844, Z -2.1667, A 0.000, B 0.000, C 0.000 }
gfCNCPoint1[23094] = {X 108.6173, Y 59.0987, Z -2.1667, A 0.000, B 0.000, C 0.000 }
gfCNCPoint1[23095] = {X 107.0213, Y 58.6267, Z -2.1667, A 0.000, B 0.000, C 0.000 }
gfCNCPoint1[23096] = {X 105.4260, Y 59.0985, Z -2.1667, A 0.000, B 0.000, C 0.000 }
gfCNCPoint1[23097] = {X 103.7872, Y 59.3842, Z -2.1667, A 0.000, B 0.000, C 0.000 }
gfCNCPoint1[23098] = {X 102.1264, Y 59.4800, Z -2.1667, A 0.000, B 0.000, C 0.000 }
gfCNCPoint1[23099] = {X 100.4656, Y 59.3847, Z -2.1667, A 0.000, B 0.000, C 0.000 }
gfCNCPoint1[23100] = {X 98.8267, Y 59.0996, Z -2.1667, A 0.000, B 0.000, C 0.000 }
gfCNCPoint1[23101] = {X 97.2313, Y 58.6283, Z -2.1667, A 0.000, B 0.000, C 0.000 }
gfCNCPoint1[23102] = {X 95.6367, Y 59.0994, Z -2.1667, A 0.000, B 0.000, C 0.000 }
gfCNCPoint1[23103] = {X 93.9986, Y 59.3845, Z -2.1667, A 0.000, B 0.000, C 0.000 }
gfCNCPoint1[23104] = {X 92.3385, Y 59.4800, Z -2.1667, A 0.000, B 0.000, C 0.000 }
gfCNCPoint1[23105] = {X 85.8951, Y 59.4800, Z -2.1667, A 0.000, B 0.000, C 0.000 }
gfCNCPoint1[23106] = {X 84.7780, Y 59.4368, Z -2.1667, A 0.000, B 0.000, C 0.000 }
gfCNCPoint1[23107] = {X 83.6677, Y 59.3077, Z -2.1667, A 0.000, B 0.000, C 0.000 }
gfCNCPoint1[23108] = {X 82.0978, Y 60.5827, Z -2.1667, A 0.000, B 0.000, C 0.000 }
gfCNCPoint1[23109] = {X 80.4031, Y 61.6862, Z -2.1667, A 0.000, B 0.000, C 0.000 }
gfCNCPoint1[23110] = {X 78.6021, Y 62.6061, Z -2.1667, A 0.000, B 0.000, C 0.000 }
gfCNCPoint1[23111] = {X 76.7146, Y 63.3324, Z -2.1667, A 0.000, B 0.000, C 0.000 }
gfCNCPoint1[23112] = {X 74.7614, Y 63.8569, Z -2.1667, A 0.000, B 0.000, C 0.000 }
gfCNCPoint1[23113] = {X 72.7640, Y 64.1739, Z -2.1667, A 0.000, B 0.000, C 0.000 }
gfCNCPoint1[23114] = {X 70.7445, Y 64.2800, Z -2.1667, A 0.000, B 0.000, C 0.000 }
gfCNCPoint1[23115] = {X 64.1851, Y 64.2800, Z -2.1667, A 0.000, B 0.000, C 0.000 }
gfCNCPoint1[23116] = {X 62.0428, Y 64.1606, Z -2.1667, A 0.000, B 0.000, C 0.000 }
gfCNCPoint1[23117] = {X 59.9269, Y 63.8039, Z -2.1667, A 0.000, B 0.000, C 0.000 }
gfCNCPoint1[23118] = {X 57.8638, Y 63.2143, Z -2.1667, A 0.000, B 0.000, C 0.000 }
gfCNCPoint1[23119] = {X 55.8790, Y 62.3991, Z -2.1667, A 0.000, B 0.000, C 0.000 }
gfCNCPoint1[23120] = {X 53.8942, Y 63.2143, Z -2.1667, A 0.000, B 0.000, C 0.000 }
gfCNCPoint1[23121] = {X 51.8311, Y 63.8039, Z -2.1667, A 0.000, B 0.000, C 0.000 }
gfCNCPoint1[23122] = {X 49.7153, Y 64.1606, Z -2.1667, A 0.000, B 0.000, C 0.000 }
gfCNCPoint1[23123] = {X 47.5729, Y 64.2800, Z -2.1667, A 0.000, B 0.000, C 0.000 }
gfCNCPoint1[23124] = {X 40.6393, Y 64.2800, Z -2.1667, A 0.000, B 0.000, C 0.000 }
gfCNCPoint1[23125] = {X 39.1545, Y 64.2227, Z -2.1667, A 0.000, B 0.000, C 0.000 }
gfCNCPoint1[23126] = {X 37.6785, Y 64.0513, Z -2.1667, A 0.000, B 0.000, C 0.000 }
gfCNCPoint1[23127] = {X 36.2201, Y 63.7667, Z -2.1667, A 0.000, B 0.000, C 0.000 }
gfCNCPoint1[23128] = {X 34.1365, Y 64.5933, Z -2.1667, A 0.000, B 0.000, C 0.000 }
gfCNCPoint1[23129] = {X 31.9839, Y 65.2187, Z -2.1667, A 0.000, B 0.000, C 0.000 }
gfCNCPoint1[23130] = {X 29.7817, Y 65.6371, Z -2.1667, A 0.000, B 0.000, C 0.000 }
gfCNCPoint1[23131] = {X 27.1137, Y 66.6851, Z -2.1667, A 0.000, B 0.000, C 0.000 }
gfCNCPoint1[23132] = {X 24.3877, Y 67.5713, Z -2.1667, A 0.000, B 0.000, C 0.000 }
gfCNCPoint1[23133] = {X 21.7651, Y 68.2576, Z -2.1667, A 0.000, B 0.000, C 0.000 }
gfCNCPoint1[23134] = {X 19.1035, Y 68.7730, Z -2.1667, A 0.000, B 0.000, C 0.000 }
gfCNCPoint1[23135] = {X 19.1035, Y 80.8949, Z -2.1667, A 0.000, B 0.000, C 0.000 }
gfCNCPoint1[23136] = {X 110.5598, Y 80.8949, Z -2.1667, A 0.000, B 0.000, C 0.000 }
gfCNCPoint1[23137] = {X 112.0540, Y 79.6756, Z -2.1667, A 0.000, B 0.000, C 0.000 }
gfCNCPoint1[23138] = {X 113.6507, Y 78.5939, Z -2.1667, A 0.000, B 0.000, C 0.000 }
gfCNCPoint1[23139] = {X 115.3372, Y 77.6584, Z -2.1667, A 0.000, B 0.000, C 0.000 }
gfCNCPoint1[23140] = {X 116.4069, Y 79.8068, Z -2.1667, A 0.000, B 0.000, C 0.000 }
gfCNCPoint1[23141] = {X 117.9835, Y 79.1080, Z -2.1667, A 0.000, B 0.000, C 0.000 }
gfCNCPoint1[23142] = {X 119.6163, Y 78.5529, Z -2.1667, A 0.000, B 0.000, C 0.000 }
gfCNCPoint1[23143] = {X 137.8578, Y 58.5211, Z -2.1667, A 0.000, B 0.000, C 0.000 }
gfCNCPoint1[23144] = {X 136.5230, Y 57.9307, Z -2.1667, A 0.000, B 0.000, C 0.000 }
gfCNCPoint1[23145] = {X 135.2543, Y 57.2090, Z -2.1667, A 0.000, B 0.000, C 0.000 }
gfCNCPoint1[23146] = {X 134.0102, Y 56.3199, Z -2.1667, A 0.000, B 0.000, C 0.000 }
gfCNCPoint1[23147] = {X 132.8669, Y 55.3046, Z -2.1667, A 0.000, B 0.000, C 0.000 }
gfCNCPoint1[23148] = {X 131.8369, Y 54.1744, Z -2.1667, A 0.000, B 0.000, C 0.000 }
gfCNCPoint1[23149] = {X 130.9319, Y 52.9419, Z -2.1667, A 0.000, B 0.000, C 0.000 }
gfCNCPoint1[23150] = {X 130.2147, Y 51.7225, Z -2.1667, A 0.000, B 0.000, C 0.000 }
gfCNCPoint1[23151] = {X 129.6199, Y 50.4390, Z -2.1667, A 0.000, B 0.000, C 0.000 }
gfCNCPoint1[23152] = {X 129.1532, Y 49.1035, Z -2.1667, A 0.000, B 0.000, C 0.000 }
gfCNCPoint1[23153] = {X 128.6036, Y 50.3877, Z -2.1667, A 0.000, B 0.000, C 0.000 }
gfCNCPoint1[23154] = {X 127.9093, Y 51.5998, Z -2.1667, A 0.000, B 0.000, C 0.000 }
gfCNCPoint1[23155] = {X 127.0798, Y 52.7237, Z -2.1667, A 0.000, B 0.000, C 0.000 }
gfCNCPoint1[23156] = {X 126.0417, Y 53.8239, Z -2.1667, A 0.000, B 0.000, C 0.000 }
gfCNCPoint1[23157] = {X 124.8743, Y 54.7858, Z -2.1667, A 0.000, B 0.000, C 0.000 }
gfCNCPoint1[23158] = {X 123.5958, Y 55.5942, Z -2.1667, A 0.000, B 0.000, C 0.000 }
gfCNCPoint1[23159] = {X 122.2263, Y 56.2365, Z -2.1667, A 0.000, B 0.000, C 0.000 }
gfCNCPoint1[23160] = {X 120.7872, Y 56.7027, Z -2.1667, A 0.000, B 0.000, C 0.000 }
gfCNCPoint1[23161] = {X 119.3012, Y 56.9853, Z -2.1667, A 0.000, B 0.000, C 0.000 }
gfCNCPoint1[23162] = {X 117.7916, Y 57.0800, Z -2.1667, A 0.000, B 0.000, C 0.000 }
gfCNCPoint1[23163] = {X 111.9185, Y 57.0800, Z -2.1667, A 0.000, B 0.000, C 0.000 }
gfCNCPoint1[23164] = {X 110.2431, Y 56.9633, Z -2.1667, A 0.000, B 0.000, C 0.000 }
gfCNCPoint1[23165] = {X 108.6001, Y 56.6153, Z -2.1667, A 0.000, B 0.000, C 0.000 }
gfCNCPoint1[23166] = {X 107.0213, Y 56.0428, Z -2.1667, A 0.000, B 0.000, C 0.000 }
gfCNCPoint1[23167] = {X 105.4432, Y 56.6151, Z -2.1667, A 0.000, B 0.000, C 0.000 }
gfCNCPoint1[23168] = {X 103.8010, Y 56.9630, Z -2.1667, A 0.000, B 0.000, C 0.000 }
gfCNCPoint1[23169] = {X 102.1265, Y 57.0800, Z -2.1667, A 0.000, B 0.000, C 0.000 }
gfCNCPoint1[23170] = {X 100.4519, Y 56.9637, Z -2.1667, A 0.000, B 0.000, C 0.000 }
gfCNCPoint1[23171] = {X 98.8096, Y 56.6164, Z -2.1667, A 0.000, B 0.000, C 0.000 }
gfCNCPoint1[23172] = {X 97.2313, Y 56.0448, Z -2.1667, A 0.000, B 0.000, C 0.000 }
gfCNCPoint1[23173] = {X 95.6538, Y 56.6162, Z -2.1667, A 0.000, B 0.000, C 0.000 }
gfCNCPoint1[23174] = {X 94.0123, Y 56.9635, Z -2.1667, A 0.000, B 0.000, C 0.000 }
gfCNCPoint1[23175] = {X 92.3385, Y 57.0800, Z -2.1667, A 0.000, B 0.000, C 0.000 }
gfCNCPoint1[23176] = {X 85.8951, Y 57.0800, Z -2.1667, A 0.000, B 0.000, C 0.000 }
gfCNCPoint1[23177] = {X 84.3894, Y 56.9858, Z -2.1667, A 0.000, B 0.000, C 0.000 }
gfCNCPoint1[23178] = {X 82.9073, Y 56.7047, Z -2.1667, A 0.000, B 0.000, C 0.000 }
gfCNCPoint1[23179] = {X 81.4846, Y 58.0224, Z -2.1667, A 0.000, B 0.000, C 0.000 }
gfCNCPoint1[23180] = {X 79.9203, Y 59.1682, Z -2.1667, A 0.000, B 0.000, C 0.000 }
gfCNCPoint1[23181] = {X 78.2348, Y 60.1271, Z -2.1667, A 0.000, B 0.000, C 0.000 }
gfCNCPoint1[23182] = {X 76.4504, Y 60.8863, Z -2.1667, A 0.000, B 0.000, C 0.000 }
gfCNCPoint1[23183] = {X 74.5908, Y 61.4359, Z -2.1667, A 0.000, B 0.000, C 0.000 }
gfCNCPoint1[23184] = {X 72.6804, Y 61.7686, Z -2.1667, A 0.000, B 0.000, C 0.000 }
gfCNCPoint1[23185] = {X 70.7445, Y 61.8800, Z -2.1667, A 0.000, B 0.000, C 0.000 }
gfCNCPoint1[23186] = {X 64.1851, Y 61.8800, Z -2.1667, A 0.000, B 0.000, C 0.000 }
gfCNCPoint1[23187] = {X 62.4514, Y 61.7907, Z -2.1667, A 0.000, B 0.000, C 0.000 }
gfCNCPoint1[23188] = {X 60.7359, Y 61.5238, Z -2.1667, A 0.000, B 0.000, C 0.000 }
gfCNCPoint1[23189] = {X 59.0570, Y 61.0822, Z -2.1667, A 0.000, B 0.000, C 0.000 }
gfCNCPoint1[23190] = {X 57.4323, Y 60.4704, Z -2.1667, A 0.000, B 0.000, C 0.000 }
gfCNCPoint1[23191] = {X 55.8790, Y 59.6950, Z -2.1667, A 0.000, B 0.000, C 0.000 }
gfCNCPoint1[23192] = {X 54.3258, Y 60.4704, Z -2.1667, A 0.000, B 0.000, C 0.000 }
gfCNCPoint1[23193] = {X 52.7011, Y 61.0822, Z -2.1667, A 0.000, B 0.000, C 0.000 }
gfCNCPoint1[23194] = {X 51.0221, Y 61.5238, Z -2.1667, A 0.000, B 0.000, C 0.000 }
gfCNCPoint1[23195] = {X 49.3067, Y 61.7907, Z -2.1667, A 0.000, B 0.000, C 0.000 }
gfCNCPoint1[23196] = {X 47.5729, Y 61.8800, Z -2.1667, A 0.000, B 0.000, C 0.000 }
gfCNCPoint1[23197] = {X 40.6393, Y 61.8800, Z -2.1667, A 0.000, B 0.000, C 0.000 }
gfCNCPoint1[23198] = {X 39.0675, Y 61.8067, Z -2.1667, A 0.000, B 0.000, C 0.000 }
gfCNCPoint1[23199] = {X 37.5094, Y 61.5873, Z -2.1667, A 0.000, B 0.000, C 0.000 }
gfCNCPoint1[23200] = {X 35.9785, Y 61.2238, Z -2.1667, A 0.000, B 0.000, C 0.000 }
gfCNCPoint1[23201] = {X 34.3397, Y 61.9593, Z -2.1667, A 0.000, B 0.000, C 0.000 }
gfCNCPoint1[23202] = {X 32.6446, Y 62.5536, Z -2.1667, A 0.000, B 0.000, C 0.000 }
gfCNCPoint1[23203] = {X 30.9054, Y 63.0023, Z -2.1667, A 0.000, B 0.000, C 0.000 }
gfCNCPoint1[23204] = {X 29.1344, Y 63.3024, Z -2.1667, A 0.000, B 0.000, C 0.000 }
gfCNCPoint1[23205] = {X 26.4534, Y 64.3720, Z -2.1667, A 0.000, B 0.000, C 0.000 }
gfCNCPoint1[23206] = {X 23.7099, Y 65.2690, Z -2.1667, A 0.000, B 0.000, C 0.000 }
gfCNCPoint1[23207] = {X 21.4042, Y 65.8780, Z -2.1667, A 0.000, B 0.000, C 0.000 }
gfCNCPoint1[23208] = {X 19.0658, Y 66.3468, Z -2.1667, A 0.000, B 0.000, C 0.000 }
gfCNCPoint1[23209] = {X 16.7035, Y 66.6737, Z -2.1667, A 0.000, B 0.000, C 0.000 }
gfCNCPoint1[23210] = {X 16.7035, Y 83.2949, Z -2.1667, A 0.000, B 0.000, C 0.000 }
gfCNCPoint1[23211] = {X 111.5064, Y 83.2949, Z -2.1667, A 0.000, B 0.000, C 0.000 }
gfCNCPoint1[23212] = {X 113.0153, Y 81.9635, Z -2.1667, A 0.000, B 0.000, C 0.000 }
gfCNCPoint1[23213] = {X 114.6547, Y 80.7965, Z -2.1667, A 0.000, B 0.000, C 0.000 }
gfCNCPoint1[23214] = {X 116.4069, Y 79.8068, Z -2.1667, A 0.000, B 0.000, C 0.000 }
gfCNCPoint1[23215] = {X 117.4766, Y 81.9553, Z -2.1667, A 0.000, B 0.000, C 0.000 }
gfCNCPoint1[23216] = {X 119.1633, Y 81.2271, Z -2.1667, A 0.000, B 0.000, C 0.000 }
gfCNCPoint1[23217] = {X 120.9192, Y 80.6866, Z -2.1667, A 0.000, B 0.000, C 0.000 }
gfCNCPoint1[23218] = {X 142.4301, Y 57.0646, Z -2.1667, A 0.000, B 0.000, C 0.000 }
gfCNCPoint1[23219] = {X 141.1670, Y 56.9340, Z -2.1667, A 0.000, B 0.000, C 0.000 }
gfCNCPoint1[23220] = {X 139.9247, Y 56.6715, Z -2.1667, A 0.000, B 0.000, C 0.000 }
gfCNCPoint1[23221] = {X 138.7167, Y 56.2800, Z -2.1667, A 0.000, B 0.000, C 0.000 }
gfCNCPoint1[23222] = {X 137.2795, Y 55.6183, Z -2.1667, A 0.000, B 0.000, C 0.000 }
gfCNCPoint1[23223] = {X 135.9412, Y 54.7744, Z -2.1667, A 0.000, B 0.000, C 0.000 }
gfCNCPoint1[23224] = {X 134.7246, Y 53.7628, Z -2.1667, A 0.000, B 0.000, C 0.000 }
gfCNCPoint1[23225] = {X 133.6507, Y 52.6009, Z -2.1667, A 0.000, B 0.000, C 0.000 }
gfCNCPoint1[23226] = {X 132.7378, Y 51.3086, Z -2.1667, A 0.000, B 0.000, C 0.000 }
gfCNCPoint1[23227] = {X 132.0016, Y 49.9081, Z -2.1667, A 0.000, B 0.000, C 0.000 }
gfCNCPoint1[23228] = {X 131.4549, Y 48.4234, Z -2.1667, A 0.000, B 0.000, C 0.000 }
gfCNCPoint1[23229] = {X 131.1845, Y 47.3200, Z -2.1667, A 0.000, B 0.000, C 0.000 }
gfCNCPoint1[23230] = {X 131.0190, Y 46.1961, Z -2.1667, A 0.000, B 0.000, C 0.000 }
gfCNCPoint1[23231] = {X 130.9598, Y 45.0616, Z -2.1667, A 0.000, B 0.000, C 0.000 }
gfCNCPoint1[23232] = {X 130.9601, Y 44.0978, Z -2.1667, A 0.000, B 0.000, C 0.000 }
gfCNCPoint1[23233] = {X 131.0921, Y 42.4244, Z -2.1667, A 0.000, B 0.000, C 0.000 }
gfCNCPoint1[23234] = {X 131.4548, Y 40.7854, Z -2.1667, A 0.000, B 0.000, C 0.000 }
gfCNCPoint1[23235] = {X 133.7565, Y 41.4655, Z -2.1667, A 0.000, B 0.000, C 0.000 }
gfCNCPoint1[23236] = {X 134.2330, Y 40.1906, Z -2.1667, A 0.000, B 0.000, C 0.000 }
gfCNCPoint1[23237] = {X 134.8836, Y 38.9952, Z -2.1667, A 0.000, B 0.000, C 0.000 }
gfCNCPoint1[23238] = {X 134.8836, Y 27.0854, Z -2.1667, A 0.000, B 0.000, C 0.000 }
gfCNCPoint1[23239] = {X 134.3931, Y 27.1259, Z -2.1667, A 0.000, B 0.000, C 0.000 }
gfCNCPoint1[23240] = {X 133.9011, Y 27.1414, Z -2.1667, A 0.000, B 0.000, C 0.000 }
gfCNCPoint1[23241] = {X 133.2006, Y 27.1415, Z -2.1667, A 0.000, B 0.000, C 0.000 }
gfCNCPoint1[23242] = {X 131.9565, Y 27.0613, Z -2.1667, A 0.000, B 0.000, C 0.000 }
gfCNCPoint1[23243] = {X 130.7330, Y 26.8217, Z -2.1667, A 0.000, B 0.000, C 0.000 }
gfCNCPoint1[23244] = {X 129.5505, Y 26.4269, Z -2.1667, A 0.000, B 0.000, C 0.000 }
gfCNCPoint1[23245] = {X 128.4284, Y 25.8834, Z -2.1667, A 0.000, B 0.000, C 0.000 }
gfCNCPoint1[23246] = {X 127.3856, Y 25.2002, Z -2.1667, A 0.000, B 0.000, C 0.000 }
gfCNCPoint1[23247] = {X 126.3438, Y 24.2943, Z -2.1667, A 0.000, B 0.000, C 0.000 }
gfCNCPoint1[23248] = {X 125.4415, Y 23.2493, Z -2.1667, A 0.000, B 0.000, C 0.000 }
gfCNCPoint1[23249] = {X 124.6971, Y 22.0867, Z -2.1667, A 0.000, B 0.000, C 0.000 }
gfCNCPoint1[23250] = {X 124.1256, Y 20.8299, Z -2.1667, A 0.000, B 0.000, C 0.000 }
gfCNCPoint1[23251] = {X 123.7387, Y 19.5046, Z -2.1667, A 0.000, B 0.000, C 0.000 }
gfCNCPoint1[23252] = {X 123.5443, Y 18.1378, Z -2.1667, A 0.000, B 0.000, C 0.000 }
gfCNCPoint1[23253] = {X 123.5432, Y 39.7459, Z -2.1667, A 0.000, B 0.000, C 0.000 }
gfCNCPoint1[23254] = {X 124.1921, Y 40.7401, Z -2.1667, A 0.000, B 0.000, C 0.000 }
gfCNCPoint1[23255] = {X 124.6707, Y 41.8265, Z -2.1667, A 0.000, B 0.000, C 0.000 }
gfCNCPoint1[23256] = {X 124.9665, Y 42.9762, Z -2.1667, A 0.000, B 0.000, C 0.000 }
gfCNCPoint1[23257] = {X 125.0714, Y 44.1587, Z -2.1667, A 0.000, B 0.000, C 0.000 }
gfCNCPoint1[23258] = {X 125.0716, Y 45.0000, Z -2.1667, A 0.000, B 0.000, C 0.000 }
gfCNCPoint1[23259] = {X 124.9610, Y 46.2642, Z -2.1667, A 0.000, B 0.000, C 0.000 }
gfCNCPoint1[23260] = {X 124.6325, Y 47.4899, Z -2.1667, A 0.000, B 0.000, C 0.000 }
gfCNCPoint1[23261] = {X 124.0962, Y 48.6400, Z -2.1667, A 0.000, B 0.000, C 0.000 }
gfCNCPoint1[23262] = {X 123.3684, Y 49.6795, Z -2.1667, A 0.000, B 0.000, C 0.000 }
gfCNCPoint1[23263] = {X 122.4711, Y 50.5768, Z -2.1667, A 0.000, B 0.000, C 0.000 }
gfCNCPoint1[23264] = {X 121.4316, Y 51.3047, Z -2.1667, A 0.000, B 0.000, C 0.000 }
gfCNCPoint1[23265] = {X 120.2815, Y 51.8410, Z -2.1667, A 0.000, B 0.000, C 0.000 }
gfCNCPoint1[23266] = {X 119.0557, Y 52.1694, Z -2.1667, A 0.000, B 0.000, C 0.000 }
gfCNCPoint1[23267] = {X 117.7916, Y 52.2800, Z -2.1667, A 0.000, B 0.000, C 0.000 }
gfCNCPoint1[23268] = {X 111.9185, Y 52.2800, Z -2.1667, A 0.000, B 0.000, C 0.000 }
gfCNCPoint1[23269] = {X 110.8481, Y 52.2009, Z -2.1667, A 0.000, B 0.000, C 0.000 }
gfCNCPoint1[23270] = {X 109.8009, Y 51.9652, Z -2.1667, A 0.000, B 0.000, C 0.000 }
gfCNCPoint1[23271] = {X 108.7998, Y 51.5782, Z -2.1667, A 0.000, B 0.000, C 0.000 }
gfCNCPoint1[23272] = {X 107.8665, Y 51.0481, Z -2.1667, A 0.000, B 0.000, C 0.000 }
gfCNCPoint1[23273] = {X 107.0213, Y 50.3866, Z -2.1667, A 0.000, B 0.000, C 0.000 }
gfCNCPoint1[23274] = {X 106.1743, Y 51.0493, Z -2.1667, A 0.000, B 0.000, C 0.000 }
gfCNCPoint1[23275] = {X 105.2389, Y 51.5800, Z -2.1667, A 0.000, B 0.000, C 0.000 }
gfCNCPoint1[23276] = {X 104.0917, Y 52.0091, Z -2.1667, A 0.000, B 0.000, C 0.000 }
gfCNCPoint1[23277] = {X 102.8887, Y 52.2397, Z -2.1667, A 0.000, B 0.000, C 0.000 }
gfCNCPoint1[23278] = {X 101.6641, Y 52.2655, Z -2.1667, A 0.000, B 0.000, C 0.000 }
gfCNCPoint1[23279] = {X 100.4526, Y 52.0855, Z -2.1667, A 0.000, B 0.000, C 0.000 }
gfCNCPoint1[23280] = {X 99.2883, Y 51.7050, Z -2.1667, A 0.000, B 0.000, C 0.000 }
gfCNCPoint1[23281] = {X 98.2043, Y 51.1347, Z -2.1667, A 0.000, B 0.000, C 0.000 }
gfCNCPoint1[23282] = {X 97.2313, Y 50.3907, Z -2.1667, A 0.000, B 0.000, C 0.000 }
gfCNCPoint1[23283] = {X 96.3865, Y 51.0508, Z -2.1667, A 0.000, B 0.000, C 0.000 }
gfCNCPoint1[23284] = {X 95.4539, Y 51.5797, Z -2.1667, A 0.000, B 0.000, C 0.000 }
gfCNCPoint1[23285] = {X 94.4538, Y 51.9659, Z -2.1667, A 0.000, B 0.000, C 0.000 }
gfCNCPoint1[23286] = {X 93.4078, Y 52.2011, Z -2.1667, A 0.000, B 0.000, C 0.000 }
gfCNCPoint1[23287] = {X 92.3385, Y 52.2800, Z -2.1667, A 0.000, B 0.000, C 0.000 }
gfCNCPoint1[23288] = {X 85.8951, Y 52.2800, Z -2.1667, A 0.000, B 0.000, C 0.000 }
gfCNCPoint1[23289] = {X 84.6852, Y 52.1788, Z -2.1667, A 0.000, B 0.000, C 0.000 }
gfCNCPoint1[23290] = {X 83.5090, Y 51.8779, Z -2.1667, A 0.000, B 0.000, C 0.000 }
gfCNCPoint1[23291] = {X 82.3992, Y 51.3857, Z -2.1667, A 0.000, B 0.000, C 0.000 }
gfCNCPoint1[23292] = {X 81.3866, Y 50.7159, Z -2.1667, A 0.000, B 0.000, C 0.000 }
gfCNCPoint1[23293] = {X 80.5223, Y 52.0937, Z -2.1667, A 0.000, B 0.000, C 0.000 }
gfCNCPoint1[23294] = {X 79.4808, Y 53.3429, Z -2.1667, A 0.000, B 0.000, C 0.000 }
gfCNCPoint1[23295] = {X 78.2809, Y 54.4408, Z -2.1667, A 0.000, B 0.000, C 0.000 }
gfCNCPoint1[23296] = {X 76.9444, Y 55.3676, Z -2.1667, A 0.000, B 0.000, C 0.000 }
gfCNCPoint1[23297] = {X 75.4955, Y 56.1065, Z -2.1667, A 0.000, B 0.000, C 0.000 }
gfCNCPoint1[23298] = {X 73.9605, Y 56.6440, Z -2.1667, A 0.000, B 0.000, C 0.000 }
gfCNCPoint1[23299] = {X 72.3672, Y 56.9705, Z -2.1667, A 0.000, B 0.000, C 0.000 }
gfCNCPoint1[23300] = {X 70.7445, Y 57.0800, Z -2.1667, A 0.000, B 0.000, C 0.000 }
gfCNCPoint1[23301] = {X 64.1851, Y 57.0800, Z -2.1667, A 0.000, B 0.000, C 0.000 }
gfCNCPoint1[23302] = {X 62.6628, Y 56.9837, Z -2.1667, A 0.000, B 0.000, C 0.000 }
gfCNCPoint1[23303] = {X 61.1646, Y 56.6963, Z -2.1667, A 0.000, B 0.000, C 0.000 }
gfCNCPoint1[23304] = {X 59.7147, Y 56.2224, Z -2.1667, A 0.000, B 0.000, C 0.000 }
gfCNCPoint1[23305] = {X 58.3360, Y 55.5695, Z -2.1667, A 0.000, B 0.000, C 0.000 }
gfCNCPoint1[23306] = {X 57.0507, Y 54.7481, Z -2.1667, A 0.000, B 0.000, C 0.000 }
gfCNCPoint1[23307] = {X 55.8790, Y 53.7713, Z -2.1667, A 0.000, B 0.000, C 0.000 }
gfCNCPoint1[23308] = {X 54.7074, Y 54.7481, Z -2.1667, A 0.000, B 0.000, C 0.000 }
gfCNCPoint1[23309] = {X 53.4220, Y 55.5695, Z -2.1667, A 0.000, B 0.000, C 0.000 }
gfCNCPoint1[23310] = {X 52.0434, Y 56.2224, Z -2.1667, A 0.000, B 0.000, C 0.000 }
gfCNCPoint1[23311] = {X 50.5934, Y 56.6963, Z -2.1667, A 0.000, B 0.000, C 0.000 }
gfCNCPoint1[23312] = {X 49.0953, Y 56.9837, Z -2.1667, A 0.000, B 0.000, C 0.000 }
gfCNCPoint1[23313] = {X 47.5729, Y 57.0800, Z -2.1667, A 0.000, B 0.000, C 0.000 }
gfCNCPoint1[23314] = {X 40.6393, Y 57.0800, Z -2.1667, A 0.000, B 0.000, C 0.000 }
gfCNCPoint1[23315] = {X 39.3237, Y 57.0081, Z -2.1667, A 0.000, B 0.000, C 0.000 }
gfCNCPoint1[23316] = {X 38.0237, Y 56.7934, Z -2.1667, A 0.000, B 0.000, C 0.000 }
gfCNCPoint1[23317] = {X 36.7549, Y 56.4384, Z -2.1667, A 0.000, B 0.000, C 0.000 }
gfCNCPoint1[23318] = {X 35.5322, Y 55.9473, Z -2.1667, A 0.000, B 0.000, C 0.000 }
gfCNCPoint1[23319] = {X 34.1219, Y 56.7816, Z -2.1667, A 0.000, B 0.000, C 0.000 }
gfCNCPoint1[23320] = {X 32.6353, Y 57.4712, Z -2.1667, A 0.000, B 0.000, C 0.000 }
gfCNCPoint1[23321] = {X 31.0875, Y 58.0091, Z -2.1667, A 0.000, B 0.000, C 0.000 }
gfCNCPoint1[23322] = {X 29.4937, Y 58.3900, Z -2.1667, A 0.000, B 0.000, C 0.000 }
gfCNCPoint1[23323] = {X 27.8699, Y 58.6102, Z -2.1667, A 0.000, B 0.000, C 0.000 }
gfCNCPoint1[23324] = {X 25.1493, Y 59.7374, Z -2.1667, A 0.000, B 0.000, C 0.000 }
gfCNCPoint1[23325] = {X 22.3542, Y 60.6644, Z -2.1667, A 0.000, B 0.000, C 0.000 }
gfCNCPoint1[23326] = {X 19.7902, Y 61.3207, Z -2.1667, A 0.000, B 0.000, C 0.000 }
gfCNCPoint1[23327] = {X 17.1836, Y 61.7797, Z -2.1667, A 0.000, B 0.000, C 0.000 }
gfCNCPoint1[23328] = {X 14.5496, Y 62.0388, Z -2.1667, A 0.000, B 0.000, C 0.000 }
gfCNCPoint1[23329] = {X 11.9035, Y 62.0964, Z -2.1667, A 0.000, B 0.000, C 0.000 }
gfCNCPoint1[23330] = {X 11.9035, Y 88.0949, Z -2.1667, A 0.000, B 0.000, C 0.000 }
gfCNCPoint1[23331] = {X 113.6338, Y 88.0949, Z -2.1667, A 0.000, B 0.000, C 0.000 }
gfCNCPoint1[23332] = {X 114.7670, Y 86.8211, Z -2.1667, A 0.000, B 0.000, C 0.000 }
gfCNCPoint1[23333] = {X 116.0422, Y 85.6893, Z -2.1667, A 0.000, B 0.000, C 0.000 }
gfCNCPoint1[23334] = {X 117.4416, Y 84.7152, Z -2.1667, A 0.000, B 0.000, C 0.000 }
gfCNCPoint1[23335] = {X 118.9457, Y 83.9124, Z -2.1667, A 0.000, B 0.000, C 0.000 }
gfCNCPoint1[23336] = {X 120.5338, Y 83.2919, Z -2.1667, A 0.000, B 0.000, C 0.000 }
gfCNCPoint1[23337] = {X 122.1838, Y 82.8624, Z -2.1667, A 0.000, B 0.000, C 0.000 }
gfCNCPoint1[23338] = {X 144.8180, Y 58.0070, Z -2.1667, A 0.000, B 0.000, C 0.000 }
gfCNCPoint1[23339] = {X 144.9143, Y 56.3323, Z -2.1667, A 0.000, B 0.000, C 0.000 }
gfCNCPoint1[23340] = {X 145.2037, Y 54.6800, Z -2.1667, A 0.000, B 0.000, C 0.000 }
gfCNCPoint1[23341] = {X 143.0396, Y 54.6800, Z -2.1667, A 0.000, B 0.000, C 0.000 }
gfCNCPoint1[23342] = {X 142.7953, Y 54.6769, Z -2.1667, A 0.000, B 0.000, C 0.000 }
gfCNCPoint1[23343] = {X 142.5512, Y 54.6677, Z -2.1667, A 0.000, B 0.000, C 0.000 }
gfCNCPoint1[23344] = {X 141.0981, Y 54.4833, Z -2.1667, A 0.000, B 0.000, C 0.000 }
gfCNCPoint1[23345] = {X 139.6895, Y 54.0818, Z -2.1667, A 0.000, B 0.000, C 0.000 }
gfCNCPoint1[23346] = {X 138.3575, Y 53.4723, Z -2.1667, A 0.000, B 0.000, C 0.000 }
gfCNCPoint1[23347] = {X 137.1328, Y 52.6689, Z -2.1667, A 0.000, B 0.000, C 0.000 }
gfCNCPoint1[23348] = {X 136.0433, Y 51.6899, Z -2.1667, A 0.000, B 0.000, C 0.000 }
gfCNCPoint1[23349] = {X 135.1140, Y 50.5576, Z -2.1667, A 0.000, B 0.000, C 0.000 }
gfCNCPoint1[23350] = {X 134.3662, Y 49.2982, Z -2.1667, A 0.000, B 0.000, C 0.000 }
gfCNCPoint1[23351] = {X 133.8170, Y 47.9403, Z -2.1667, A 0.000, B 0.000, C 0.000 }
gfCNCPoint1[23352] = {X 133.4789, Y 46.5151, Z -2.1667, A 0.000, B 0.000, C 0.000 }
gfCNCPoint1[23353] = {X 133.3598, Y 45.0552, Z -2.1667, A 0.000, B 0.000, C 0.000 }
gfCNCPoint1[23354] = {X 133.3601, Y 44.1104, Z -2.1667, A 0.000, B 0.000, C 0.000 }
gfCNCPoint1[23355] = {X 133.4665, Y 42.7742, Z -2.1667, A 0.000, B 0.000, C 0.000 }
gfCNCPoint1[23356] = {X 133.7565, Y 41.4655, Z -2.1667, A 0.000, B 0.000, C 0.000 }
gfCNCPoint1[23357] = {X 136.0581, Y 42.1457, Z -2.1667, A 0.000, B 0.000, C 0.000 }
gfCNCPoint1[23358] = {X 136.3664, Y 41.2990, Z -2.1667, A 0.000, B 0.000, C 0.000 }
gfCNCPoint1[23359] = {X 136.7770, Y 40.4969, Z -2.1667, A 0.000, B 0.000, C 0.000 }
gfCNCPoint1[23360] = {X 137.2836, Y 39.7516, Z -2.1667, A 0.000, B 0.000, C 0.000 }
gfCNCPoint1[23361] = {X 137.2836, Y 23.8768, Z -2.1667, A 0.000, B 0.000, C 0.000 }
gfCNCPoint1[23362] = {X 136.4352, Y 24.2641, Z -2.1667, A 0.000, B 0.000, C 0.000 }
gfCNCPoint1[23363] = {X 135.5443, Y 24.5398, Z -2.1667, A 0.000, B 0.000, C 0.000 }
gfCNCPoint1[23364] = {X 134.6254, Y 24.6993, Z -2.1667, A 0.000, B 0.000, C 0.000 }
gfCNCPoint1[23365] = {X 134.2595, Y 24.7296, Z -2.1667, A 0.000, B 0.000, C 0.000 }
gfCNCPoint1[23366] = {X 133.8926, Y 24.7414, Z -2.1667, A 0.000, B 0.000, C 0.000 }
gfCNCPoint1[23367] = {X 133.2006, Y 24.7415, Z -2.1667, A 0.000, B 0.000, C 0.000 }
gfCNCPoint1[23368] = {X 131.9922, Y 24.6405, Z -2.1667, A 0.000, B 0.000, C 0.000 }
gfCNCPoint1[23369] = {X 130.8173, Y 24.3404, Z -2.1667, A 0.000, B 0.000, C 0.000 }
gfCNCPoint1[23370] = {X 129.7086, Y 23.8493, Z -2.1667, A 0.000, B 0.000, C 0.000 }
gfCNCPoint1[23371] = {X 128.6967, Y 23.1810, Z -2.1667, A 0.000, B 0.000, C 0.000 }
gfCNCPoint1[23372] = {X 127.8098, Y 22.3541, Z -2.1667, A 0.000, B 0.000, C 0.000 }
gfCNCPoint1[23373] = {X 127.0724, Y 21.3914, Z -2.1667, A 0.000, B 0.000, C 0.000 }
gfCNCPoint1[23374] = {X 126.5051, Y 20.3196, Z -2.1667, A 0.000, B 0.000, C 0.000 }
gfCNCPoint1[23375] = {X 126.1236, Y 19.1685, Z -2.1667, A 0.000, B 0.000, C 0.000 }
gfCNCPoint1[23376] = {X 125.9384, Y 17.9701, Z -2.1667, A 0.000, B 0.000, C 0.000 }
gfCNCPoint1[23377] = {X 125.9251, Y 17.7160, Z -2.1667, A 0.000, B 0.000, C 0.000 }
gfCNCPoint1[23378] = {X 125.9206, Y 17.4615, Z -2.1667, A 0.000, B 0.000, C 0.000 }
gfCNCPoint1[23379] = {X 125.9206, Y 10.4835, Z -2.1667, A 0.000, B 0.000, C 0.000 }
gfCNCPoint1[23380] = {X 125.9372, Y 9.9932, Z -2.1667, A 0.000, B 0.000, C 0.000 }
gfCNCPoint1[23381] = {X 125.9867, Y 9.5051, Z -2.1667, A 0.000, B 0.000, C 0.000 }
gfCNCPoint1[23382] = {X 121.8687, Y 9.5051, Z -2.1667, A 0.000, B 0.000, C 0.000 }
gfCNCPoint1[23383] = {X 122.3091, Y 10.3411, Z -2.1667, A 0.000, B 0.000, C 0.000 }
gfCNCPoint1[23384] = {X 122.5801, Y 11.2463, Z -2.1667, A 0.000, B 0.000, C 0.000 }
gfCNCPoint1[23385] = {X 122.6716, Y 12.1868, Z -2.1667, A 0.000, B 0.000, C 0.000 }
gfCNCPoint1[23386] = {X 122.6714, Y 13.0237, Z -2.1667, A 0.000, B 0.000, C 0.000 }
gfCNCPoint1[23387] = {X 122.5640, Y 13.9971, Z -2.1667, A 0.000, B 0.000, C 0.000 }
gfCNCPoint1[23388] = {X 122.2645, Y 14.9294, Z -2.1667, A 0.000, B 0.000, C 0.000 }
gfCNCPoint1[23389] = {X 121.7848, Y 15.7831, Z -2.1667, A 0.000, B 0.000, C 0.000 }
gfCNCPoint1[23390] = {X 121.1444, Y 16.5239, Z -2.1667, A 0.000, B 0.000, C 0.000 }
gfCNCPoint1[23391] = {X 121.1432, Y 40.6618, Z -2.1667, A 0.000, B 0.000, C 0.000 }
gfCNCPoint1[23392] = {X 121.7849, Y 41.4039, Z -2.1667, A 0.000, B 0.000, C 0.000 }
gfCNCPoint1[23393] = {X 122.2653, Y 42.2593, Z -2.1667, A 0.000, B 0.000, C 0.000 }
gfCNCPoint1[23394] = {X 122.5648, Y 43.1935, Z -2.1667, A 0.000, B 0.000, C 0.000 }
gfCNCPoint1[23395] = {X 122.6714, Y 44.1688, Z -2.1667, A 0.000, B 0.000, C 0.000 }
gfCNCPoint1[23396] = {X 122.6716, Y 45.0000, Z -2.1667, A 0.000, B 0.000, C 0.000 }
gfCNCPoint1[23397] = {X 122.5778, Y 45.9520, Z -2.1667, A 0.000, B 0.000, C 0.000 }
gfCNCPoint1[23398] = {X 122.3001, Y 46.8675, Z -2.1667, A 0.000, B 0.000, C 0.000 }
gfCNCPoint1[23399] = {X 121.8491, Y 47.7112, Z -2.1667, A 0.000, B 0.000, C 0.000 }
gfCNCPoint1[23400] = {X 121.2423, Y 48.4507, Z -2.1667, A 0.000, B 0.000, C 0.000 }
gfCNCPoint1[23401] = {X 120.5028, Y 49.0576, Z -2.1667, A 0.000, B 0.000, C 0.000 }
gfCNCPoint1[23402] = {X 119.6591, Y 49.5085, Z -2.1667, A 0.000, B 0.000, C 0.000 }
gfCNCPoint1[23403] = {X 118.7436, Y 49.7862, Z -2.1667, A 0.000, B 0.000, C 0.000 }
gfCNCPoint1[23404] = {X 117.7916, Y 49.8800, Z -2.1667, A 0.000, B 0.000, C 0.000 }
gfCNCPoint1[23405] = {X 111.9185, Y 49.8800, Z -2.1667, A 0.000, B 0.000, C 0.000 }
gfCNCPoint1[23406] = {X 111.0234, Y 49.7972, Z -2.1667, A 0.000, B 0.000, C 0.000 }
gfCNCPoint1[23407] = {X 110.1587, Y 49.5517, Z -2.1667, A 0.000, B 0.000, C 0.000 }
gfCNCPoint1[23408] = {X 109.3537, Y 49.1517, Z -2.1667, A 0.000, B 0.000, C 0.000 }
gfCNCPoint1[23409] = {X 108.6357, Y 48.6108, Z -2.1667, A 0.000, B 0.000, C 0.000 }
gfCNCPoint1[23410] = {X 108.0714, Y 48.0024, Z -2.1667, A 0.000, B 0.000, C 0.000 }
gfCNCPoint1[23411] = {X 107.6183, Y 47.3071, Z -2.1667, A 0.000, B 0.000, C 0.000 }
gfCNCPoint1[23412] = {X 107.2895, Y 46.5451, Z -2.1667, A 0.000, B 0.000, C 0.000 }
gfCNCPoint1[23413] = {X 107.0947, Y 45.7384, Z -2.1667, A 0.000, B 0.000, C 0.000 }
gfCNCPoint1[23414] = {X 106.6287, Y 46.8768, Z -2.1667, A 0.000, B 0.000, C 0.000 }
gfCNCPoint1[23415] = {X 106.1131, Y 47.8110, Z -2.1667, A 0.000, B 0.000, C 0.000 }
gfCNCPoint1[23416] = {X 105.4068, Y 48.6108, Z -2.1667, A 0.000, B 0.000, C 0.000 }
gfCNCPoint1[23417] = {X 104.8391, Y 49.0550, Z -2.1667, A 0.000, B 0.000, C 0.000 }
gfCNCPoint1[23418] = {X 104.2121, Y 49.4107, Z -2.1667, A 0.000, B 0.000, C 0.000 }
gfCNCPoint1[23419] = {X 103.3106, Y 49.7335, Z -2.1667, A 0.000, B 0.000, C 0.000 }
gfCNCPoint1[23420] = {X 102.3635, Y 49.8741, Z -2.1667, A 0.000, B 0.000, C 0.000 }
gfCNCPoint1[23421] = {X 101.4071, Y 49.8271, Z -2.1667, A 0.000, B 0.000, C 0.000 }
gfCNCPoint1[23422] = {X 100.4784, Y 49.5941, Z -2.1667, A 0.000, B 0.000, C 0.000 }
gfCNCPoint1[23423] = {X 99.6130, Y 49.1844, Z -2.1667, A 0.000, B 0.000, C 0.000 }
gfCNCPoint1[23424] = {X 98.8443, Y 48.6135, Z -2.1667, A 0.000, B 0.000, C 0.000 }
gfCNCPoint1[23425] = {X 98.1362, Y 47.8127, Z -2.1667, A 0.000, B 0.000, C 0.000 }
gfCNCPoint1[23426] = {X 97.6194, Y 46.8769, Z -2.1667, A 0.000, B 0.000, C 0.000 }
gfCNCPoint1[23427] = {X 97.1600, Y 45.7536, Z -2.1667, A 0.000, B 0.000, C 0.000 }
gfCNCPoint1[23428] = {X 96.9635, Y 46.5570, Z -2.1667, A 0.000, B 0.000, C 0.000 }
gfCNCPoint1[23429] = {X 96.6342, Y 47.3156, Z -2.1667, A 0.000, B 0.000, C 0.000 }
gfCNCPoint1[23430] = {X 96.1814, Y 48.0078, Z -2.1667, A 0.000, B 0.000, C 0.000 }
gfCNCPoint1[23431] = {X 95.6183, Y 48.6135, Z -2.1667, A 0.000, B 0.000, C 0.000 }
gfCNCPoint1[23432] = {X 94.9007, Y 49.1533, Z -2.1667, A 0.000, B 0.000, C 0.000 }
gfCNCPoint1[23433] = {X 94.0964, Y 49.5524, Z -2.1667, A 0.000, B 0.000, C 0.000 }
gfCNCPoint1[23434] = {X 93.2326, Y 49.7974, Z -2.1667, A 0.000, B 0.000, C 0.000 }
gfCNCPoint1[23435] = {X 92.3385, Y 49.8800, Z -2.1667, A 0.000, B 0.000, C 0.000 }
gfCNCPoint1[23436] = {X 85.8951, Y 49.8800, Z -2.1667, A 0.000, B 0.000, C 0.000 }
gfCNCPoint1[23437] = {X 85.0841, Y 49.8121, Z -2.1667, A 0.000, B 0.000, C 0.000 }
gfCNCPoint1[23438] = {X 84.2956, Y 49.6104, Z -2.1667, A 0.000, B 0.000, C 0.000 }
gfCNCPoint1[23439] = {X 83.5517, Y 49.2805, Z -2.1667, A 0.000, B 0.000, C 0.000 }
gfCNCPoint1[23440] = {X 82.8729, Y 48.8316, Z -2.1667, A 0.000, B 0.000, C 0.000 }
gfCNCPoint1[23441] = {X 82.2391, Y 48.2324, Z -2.1667, A 0.000, B 0.000, C 0.000 }
gfCNCPoint1[23442] = {X 81.7221, Y 47.5300, Z -2.1667, A 0.000, B 0.000, C 0.000 }
gfCNCPoint1[23443] = {X 81.3384, Y 46.7467, Z -2.1667, A 0.000, B 0.000, C 0.000 }
gfCNCPoint1[23444] = {X 81.1002, Y 45.9077, Z -2.1667, A 0.000, B 0.000, C 0.000 }
gfCNCPoint1[23445] = {X 81.0152, Y 45.0397, Z -2.1667, A 0.000, B 0.000, C 0.000 }
gfCNCPoint1[23446] = {X 81.0151, Y 44.2032, Z -2.1667, A 0.000, B 0.000, C 0.000 }
gfCNCPoint1[23447] = {X 81.1205, Y 43.2197, Z -2.1667, A 0.000, B 0.000, C 0.000 }
gfCNCPoint1[23448] = {X 81.4196, Y 42.2770, Z -2.1667, A 0.000, B 0.000, C 0.000 }
gfCNCPoint1[23449] = {X 81.9004, Y 41.4126, Z -2.1667, A 0.000, B 0.000, C 0.000 }
gfCNCPoint1[23450] = {X 82.5437, Y 40.6614, Z -2.1667, A 0.000, B 0.000, C 0.000 }
gfCNCPoint1[23451] = {X 82.5435, Y 25.2487, Z -2.1667, A 0.000, B 0.000, C 0.000 }
gfCNCPoint1[23452] = {X 77.7435, Y 25.2488, Z -2.1667, A 0.000, B 0.000, C 0.000 }
gfCNCPoint1[23453] = {X 77.7434, Y 18.1985, Z -2.1667, A 0.000, B 0.000, C 0.000 }
gfCNCPoint1[23454] = {X 77.0785, Y 16.9744, Z -2.1667, A 0.000, B 0.000, C 0.000 }
gfCNCPoint1[23455] = {X 76.5962, Y 15.6676, Z -2.1667, A 0.000, B 0.000, C 0.000 }
gfCNCPoint1[23456] = {X 76.3065, Y 14.3051, Z -2.1667, A 0.000, B 0.000, C 0.000 }
gfCNCPoint1[23457] = {X 74.0412, Y 14.3051, Z -2.1667, A 0.000, B 0.000, C 0.000 }
gfCNCPoint1[23458] = {X 73.9997, Y 14.6973, Z -2.1667, A 0.000, B 0.000, C 0.000 }
gfCNCPoint1[23459] = {X 73.9475, Y 15.0883, Z -2.1667, A 0.000, B 0.000, C 0.000 }
gfCNCPoint1[23460] = {X 77.7435, Y 25.2488, Z -2.1667, A 0.000, B 0.000, C 0.000 }
gfCNCPoint1[23461] = {X 80.1435, Y 25.2488, Z -2.1667, A 0.000, B 0.000, C 0.000 }
gfCNCPoint1[23462] = {X 80.1434, Y 17.4409, Z -2.1667, A 0.000, B 0.000, C 0.000 }
gfCNCPoint1[23463] = {X 79.4948, Y 16.4472, Z -2.1667, A 0.000, B 0.000, C 0.000 }
gfCNCPoint1[23464] = {X 79.0162, Y 15.3613, Z -2.1667, A 0.000, B 0.000, C 0.000 }
gfCNCPoint1[23465] = {X 78.7204, Y 14.2121, Z -2.1667, A 0.000, B 0.000, C 0.000 }
gfCNCPoint1[23466] = {X 78.6153, Y 13.0301, Z -2.1667, A 0.000, B 0.000, C 0.000 }
gfCNCPoint1[23467] = {X 78.6151, Y 12.1868, Z -2.1667, A 0.000, B 0.000, C 0.000 }
gfCNCPoint1[23468] = {X 78.6164, Y 12.0459, Z -2.1667, A 0.000, B 0.000, C 0.000 }
gfCNCPoint1[23469] = {X 78.6205, Y 11.9051, Z -2.1667, A 0.000, B 0.000, C 0.000 }
gfCNCPoint1[23470] = {X 71.6988, Y 11.9051, Z -2.1667, A 0.000, B 0.000, C 0.000 }
gfCNCPoint1[23471] = {X 71.7013, Y 12.0459, Z -2.1667, A 0.000, B 0.000, C 0.000 }
gfCNCPoint1[23472] = {X 71.7021, Y 12.1868, Z -2.1667, A 0.000, B 0.000, C 0.000 }
gfCNCPoint1[23473] = {X 71.7016, Y 13.0911, Z -2.1667, A 0.000, B 0.000, C 0.000 }
gfCNCPoint1[23474] = {X 71.6390, Y 14.2116, Z -2.1667, A 0.000, B 0.000, C 0.000 }
gfCNCPoint1[23475] = {X 71.4726, Y 15.3215, Z -2.1667, A 0.000, B 0.000, C 0.000 }
gfCNCPoint1[23476] = {X 78.9544, Y 35.3474, Z -2.1667, A 0.000, B 0.000, C 0.000 }
gfCNCPoint1[23477] = {X 79.5720, Y 35.9625, Z -2.1667, A 0.000, B 0.000, C 0.000 }
gfCNCPoint1[23478] = {X 80.1437, Y 36.6205, Z -2.1667, A 0.000, B 0.000, C 0.000 }
gfCNCPoint1[23479] = {X 80.1435, Y 25.2488, Z -2.1667, A 0.000, B 0.000, C 0.000 }
gfCNCPoint1[23480] = {X 82.5435, Y 25.2487, Z -2.1667, A 0.000, B 0.000, C 0.000 }
gfCNCPoint1[23481] = {X 82.5434, Y 16.5250, Z -2.1667, A 0.000, B 0.000, C 0.000 }
gfCNCPoint1[23482] = {X 81.9019, Y 15.7832, Z -2.1667, A 0.000, B 0.000, C 0.000 }
gfCNCPoint1[23483] = {X 81.4217, Y 14.9282, Z -2.1667, A 0.000, B 0.000, C 0.000 }
gfCNCPoint1[23484] = {X 81.1221, Y 13.9944, Z -2.1667, A 0.000, B 0.000, C 0.000 }
gfCNCPoint1[23485] = {X 81.0153, Y 13.0196, Z -2.1667, A 0.000, B 0.000, C 0.000 }
gfCNCPoint1[23486] = {X 81.0151, Y 12.1868, Z -2.1667, A 0.000, B 0.000, C 0.000 }
gfCNCPoint1[23487] = {X 81.0160, Y 12.0924, Z -2.1667, A 0.000, B 0.000, C 0.000 }
gfCNCPoint1[23488] = {X 81.0187, Y 11.9980, Z -2.1667, A 0.000, B 0.000, C 0.000 }
gfCNCPoint1[23489] = {X 81.1324, Y 11.1231, Z -2.1667, A 0.000, B 0.000, C 0.000 }
gfCNCPoint1[23490] = {X 81.4018, Y 10.2830, Z -2.1667, A 0.000, B 0.000, C 0.000 }
gfCNCPoint1[23491] = {X 81.8180, Y 9.5051, Z -2.1667, A 0.000, B 0.000, C 0.000 }
gfCNCPoint1[23492] = {X 82.2190, Y 9.7689, Z -2.1667, A 0.000, B 0.000, C 0.000 }
gfCNCPoint1[23493] = {X 82.7658, Y 9.0936, Z -2.1667, A 0.000, B 0.000, C 0.000 }
gfCNCPoint1[23494] = {X 83.4347, Y 8.5390, Z -2.1667, A 0.000, B 0.000, C 0.000 }
gfCNCPoint1[23495] = {X 84.1995, Y 8.1266, Z -2.1667, A 0.000, B 0.000, C 0.000 }
gfCNCPoint1[23496] = {X 85.0304, Y 7.8726, Z -2.1667, A 0.000, B 0.000, C 0.000 }
gfCNCPoint1[23497] = {X 85.8951, Y 7.7868, Z -2.1667, A 0.000, B 0.000, C 0.000 }
gfCNCPoint1[23498] = {X 94.0497, Y 7.7868, Z -2.1667, A 0.000, B 0.000, C 0.000 }
gfCNCPoint1[23499] = {X 95.0288, Y 7.8971, Z -2.1667, A 0.000, B 0.000, C 0.000 }
gfCNCPoint1[23500] = {X 95.9588, Y 8.2226, Z -2.1667, A 0.000, B 0.000, C 0.000 }
gfCNCPoint1[23501] = {X 96.7930, Y 8.7468, Z -2.1667, A 0.000, B 0.000, C 0.000 }
gfCNCPoint1[23502] = {X 97.4897, Y 9.4435, Z -2.1667, A 0.000, B 0.000, C 0.000 }
gfCNCPoint1[23503] = {X 98.0139, Y 10.2777, Z -2.1667, A 0.000, B 0.000, C 0.000 }
gfCNCPoint1[23504] = {X 98.3394, Y 11.2077, Z -2.1667, A 0.000, B 0.000, C 0.000 }
gfCNCPoint1[23505] = {X 98.4497, Y 12.1868, Z -2.1667, A 0.000, B 0.000, C 0.000 }
gfCNCPoint1[23506] = {X 98.4494, Y 13.0233, Z -2.1667, A 0.000, B 0.000, C 0.000 }
gfCNCPoint1[23507] = {X 98.3723, Y 13.7995, Z -2.1667, A 0.000, B 0.000, C 0.000 }
gfCNCPoint1[23508] = {X 98.1593, Y 14.5499, Z -2.1667, A 0.000, B 0.000, C 0.000 }
gfCNCPoint1[23509] = {X 97.8172, Y 15.2509, Z -2.1667, A 0.000, B 0.000, C 0.000 }
gfCNCPoint1[23510] = {X 98.3668, Y 16.6193, Z -2.1667, A 0.000, B 0.000, C 0.000 }
gfCNCPoint1[23511] = {X 101.8765, Y 25.3192, Z -2.1667, A 0.000, B 0.000, C 0.000 }
gfCNCPoint1[23512] = {X 105.9246, Y 15.2238, Z -2.1667, A 0.000, B 0.000, C 0.000 }
gfCNCPoint1[23513] = {X 105.5858, Y 14.5161, Z -2.1667, A 0.000, B 0.000, C 0.000 }
gfCNCPoint1[23514] = {X 105.3782, Y 13.7594, Z -2.1667, A 0.000, B 0.000, C 0.000 }
gfCNCPoint1[23515] = {X 105.3083, Y 12.9779, Z -2.1667, A 0.000, B 0.000, C 0.000 }
gfCNCPoint1[23516] = {X 105.3083, Y 12.1868, Z -2.1667, A 0.000, B 0.000, C 0.000 }
gfCNCPoint1[23517] = {X 105.4186, Y 11.2077, Z -2.1667, A 0.000, B 0.000, C 0.000 }
gfCNCPoint1[23518] = {X 105.7440, Y 10.2777, Z -2.1667, A 0.000, B 0.000, C 0.000 }
gfCNCPoint1[23519] = {X 106.2682, Y 9.4435, Z -2.1667, A 0.000, B 0.000, C 0.000 }
gfCNCPoint1[23520] = {X 106.9649, Y 8.7468, Z -2.1667, A 0.000, B 0.000, C 0.000 }
gfCNCPoint1[23521] = {X 107.7992, Y 8.2226, Z -2.1667, A 0.000, B 0.000, C 0.000 }
gfCNCPoint1[23522] = {X 108.7292, Y 7.8971, Z -2.1667, A 0.000, B 0.000, C 0.000 }
gfCNCPoint1[23523] = {X 109.7083, Y 7.7868, Z -2.1667, A 0.000, B 0.000, C 0.000 }
gfCNCPoint1[23524] = {X 117.7916, Y 7.7868, Z -2.1667, A 0.000, B 0.000, C 0.000 }
gfCNCPoint1[23525] = {X 118.7707, Y 7.8971, Z -2.1667, A 0.000, B 0.000, C 0.000 }
gfCNCPoint1[23526] = {X 119.7007, Y 8.2226, Z -2.1667, A 0.000, B 0.000, C 0.000 }
gfCNCPoint1[23527] = {X 120.5349, Y 8.7468, Z -2.1667, A 0.000, B 0.000, C 0.000 }
gfCNCPoint1[23528] = {X 121.2316, Y 9.4435, Z -2.1667, A 0.000, B 0.000, C 0.000 }
gfCNCPoint1[23529] = {X 121.7558, Y 10.2777, Z -2.1667, A 0.000, B 0.000, C 0.000 }
gfCNCPoint1[23530] = {X 122.0813, Y 11.2077, Z -2.1667, A 0.000, B 0.000, C 0.000 }
gfCNCPoint1[23531] = {X 122.1916, Y 12.1868, Z -2.1667, A 0.000, B 0.000, C 0.000 }
gfCNCPoint1[23532] = {X 122.1913, Y 13.0233, Z -2.1667, A 0.000, B 0.000, C 0.000 }
gfCNCPoint1[23533] = {X 122.0830, Y 13.9492, Z -2.1667, A 0.000, B 0.000, C 0.000 }
gfCNCPoint1[23534] = {X 121.7821, Y 14.8316, Z -2.1667, A 0.000, B 0.000, C 0.000 }
gfCNCPoint1[23535] = {X 121.3020, Y 15.6307, Z -2.1667, A 0.000, B 0.000, C 0.000 }
gfCNCPoint1[23536] = {X 120.6644, Y 16.3107, Z -2.1667, A 0.000, B 0.000, C 0.000 }
gfCNCPoint1[23537] = {X 120.6631, Y 40.8755, Z -2.1667, A 0.000, B 0.000, C 0.000 }
gfCNCPoint1[23538] = {X 120.6784, Y 40.8882, Z -2.1667, A 0.000, B 0.000, C 0.000 }
gfCNCPoint1[23539] = {X 121.3172, Y 41.5763, Z -2.1667, A 0.000, B 0.000, C 0.000 }
gfCNCPoint1[23540] = {X 121.7955, Y 42.3843, Z -2.1667, A 0.000, B 0.000, C 0.000 }
gfCNCPoint1[23541] = {X 122.0914, Y 43.2754, Z -2.1667, A 0.000, B 0.000, C 0.000 }
gfCNCPoint1[23542] = {X 122.1916, Y 44.2089, Z -2.1667, A 0.000, B 0.000, C 0.000 }
gfCNCPoint1[23543] = {X 122.1916, Y 45.0000, Z -2.1667, A 0.000, B 0.000, C 0.000 }
gfCNCPoint1[23544] = {X 122.0813, Y 45.9791, Z -2.1667, A 0.000, B 0.000, C 0.000 }
gfCNCPoint1[23545] = {X 121.7558, Y 46.9091, Z -2.1667, A 0.000, B 0.000, C 0.000 }
gfCNCPoint1[23546] = {X 121.2316, Y 47.7434, Z -2.1667, A 0.000, B 0.000, C 0.000 }
gfCNCPoint1[23547] = {X 120.5349, Y 48.4401, Z -2.1667, A 0.000, B 0.000, C 0.000 }
gfCNCPoint1[23548] = {X 119.7007, Y 48.9643, Z -2.1667, A 0.000, B 0.000, C 0.000 }
gfCNCPoint1[23549] = {X 118.7707, Y 49.2897, Z -2.1667, A 0.000, B 0.000, C 0.000 }
gfCNCPoint1[23550] = {X 117.7916, Y 49.4000, Z -2.1667, A 0.000, B 0.000, C 0.000 }
gfCNCPoint1[23551] = {X 111.9185, Y 49.4000, Z -2.1667, A 0.000, B 0.000, C 0.000 }
gfCNCPoint1[23552] = {X 110.9394, Y 49.2897, Z -2.1667, A 0.000, B 0.000, C 0.000 }
gfCNCPoint1[23553] = {X 110.0094, Y 48.9643, Z -2.1667, A 0.000, B 0.000, C 0.000 }
gfCNCPoint1[23554] = {X 109.1751, Y 48.4400, Z -2.1667, A 0.000, B 0.000, C 0.000 }
gfCNCPoint1[23555] = {X 108.4784, Y 47.7433, Z -2.1667, A 0.000, B 0.000, C 0.000 }
gfCNCPoint1[23556] = {X 107.9542, Y 46.9091, Z -2.1667, A 0.000, B 0.000, C 0.000 }
gfCNCPoint1[23557] = {X 107.6288, Y 45.9791, Z -2.1667, A 0.000, B 0.000, C 0.000 }
gfCNCPoint1[23558] = {X 107.5185, Y 45.0000, Z -2.1667, A 0.000, B 0.000, C 0.000 }
gfCNCPoint1[23559] = {X 107.5185, Y 44.1778, Z -2.1667, A 0.000, B 0.000, C 0.000 }
gfCNCPoint1[23560] = {X 107.5548, Y 43.6249, Z -2.1667, A 0.000, B 0.000, C 0.000 }
gfCNCPoint1[23561] = {X 107.6633, Y 43.0815, Z -2.1667, A 0.000, B 0.000, C 0.000 }
gfCNCPoint1[23562] = {X 106.1856, Y 46.6923, Z -2.1667, A 0.000, B 0.000, C 0.000 }
gfCNCPoint1[23563] = {X 105.8087, Y 47.4049, Z -2.1667, A 0.000, B 0.000, C 0.000 }
gfCNCPoint1[23564] = {X 105.3081, Y 48.0367, Z -2.1667, A 0.000, B 0.000, C 0.000 }
gfCNCPoint1[23565] = {X 104.7006, Y 48.5667, Z -2.1667, A 0.000, B 0.000, C 0.000 }
gfCNCPoint1[23566] = {X 104.0067, Y 48.9769, Z -2.1667, A 0.000, B 0.000, C 0.000 }
gfCNCPoint1[23567] = {X 103.0414, Y 49.3033, Z -2.1667, A 0.000, B 0.000, C 0.000 }
gfCNCPoint1[23568] = {X 102.0269, Y 49.3989, Z -2.1667, A 0.000, B 0.000, C 0.000 }
gfCNCPoint1[23569] = {X 101.0176, Y 49.2586, Z -2.1667, A 0.000, B 0.000, C 0.000 }
gfCNCPoint1[23570] = {X 100.0676, Y 48.8899, Z -2.1667, A 0.000, B 0.000, C 0.000 }
gfCNCPoint1[23571] = {X 99.2280, Y 48.3125, Z -2.1667, A 0.000, B 0.000, C 0.000 }
gfCNCPoint1[23572] = {X 98.5436, Y 47.5575, Z -2.1667, A 0.000, B 0.000, C 0.000 }
gfCNCPoint1[23573] = {X 98.0514, Y 46.6653, Z -2.1667, A 0.000, B 0.000, C 0.000 }
gfCNCPoint1[23574] = {X 96.5855, Y 43.0802, Z -2.1667, A 0.000, B 0.000, C 0.000 }
gfCNCPoint1[23575] = {X 96.6980, Y 43.6397, Z -2.1667, A 0.000, B 0.000, C 0.000 }
gfCNCPoint1[23576] = {X 96.7385, Y 44.2089, Z -2.1667, A 0.000, B 0.000, C 0.000 }
gfCNCPoint1[23577] = {X 96.7383, Y 45.0423, Z -2.1667, A 0.000, B 0.000, C 0.000 }
gfCNCPoint1[23578] = {X 96.6200, Y 46.0144, Z -2.1667, A 0.000, B 0.000, C 0.000 }
gfCNCPoint1[23579] = {X 96.2896, Y 46.9363, Z -2.1667, A 0.000, B 0.000, C 0.000 }
gfCNCPoint1[23580] = {X 95.7635, Y 47.7622, Z -2.1667, A 0.000, B 0.000, C 0.000 }
gfCNCPoint1[23581] = {X 95.0677, Y 48.4513, Z -2.1667, A 0.000, B 0.000, C 0.000 }
gfCNCPoint1[23582] = {X 94.2367, Y 48.9695, Z -2.1667, A 0.000, B 0.000, C 0.000 }
gfCNCPoint1[23583] = {X 93.3117, Y 49.2910, Z -2.1667, A 0.000, B 0.000, C 0.000 }
gfCNCPoint1[23584] = {X 92.3385, Y 49.4000, Z -2.1667, A 0.000, B 0.000, C 0.000 }
gfCNCPoint1[23585] = {X 85.8951, Y 49.4000, Z -2.1667, A 0.000, B 0.000, C 0.000 }
gfCNCPoint1[23586] = {X 84.9160, Y 49.2897, Z -2.1667, A 0.000, B 0.000, C 0.000 }
gfCNCPoint1[23587] = {X 83.9860, Y 48.9643, Z -2.1667, A 0.000, B 0.000, C 0.000 }
gfCNCPoint1[23588] = {X 83.1517, Y 48.4400, Z -2.1667, A 0.000, B 0.000, C 0.000 }
gfCNCPoint1[23589] = {X 82.4550, Y 47.7433, Z -2.1667, A 0.000, B 0.000, C 0.000 }
gfCNCPoint1[23590] = {X 81.9308, Y 46.9091, Z -2.1667, A 0.000, B 0.000, C 0.000 }
gfCNCPoint1[23591] = {X 81.6054, Y 45.9791, Z -2.1667, A 0.000, B 0.000, C 0.000 }
gfCNCPoint1[23592] = {X 81.4951, Y 45.0000, Z -2.1667, A 0.000, B 0.000, C 0.000 }
gfCNCPoint1[23593] = {X 81.4951, Y 44.2063, Z -2.1667, A 0.000, B 0.000, C 0.000 }
gfCNCPoint1[23594] = {X 81.6008, Y 43.2692, Z -2.1667, A 0.000, B 0.000, C 0.000 }
gfCNCPoint1[23595] = {X 81.9011, Y 42.3753, Z -2.1667, A 0.000, B 0.000, C 0.000 }
gfCNCPoint1[23596] = {X 82.3826, Y 41.5645, Z -2.1667, A 0.000, B 0.000, C 0.000 }
gfCNCPoint1[23597] = {X 83.0237, Y 40.8729, Z -2.1667, A 0.000, B 0.000, C 0.000 }
gfCNCPoint1[23598] = {X 83.0234, Y 16.3117, Z -2.1667, A 0.000, B 0.000, C 0.000 }
gfCNCPoint1[23599] = {X 82.3785, Y 15.6225, Z -2.1667, A 0.000, B 0.000, C 0.000 }
gfCNCPoint1[23600] = {X 81.8953, Y 14.8116, Z -2.1667, A 0.000, B 0.000, C 0.000 }
gfCNCPoint1[23601] = {X 81.5963, Y 13.9164, Z -2.1667, A 0.000, B 0.000, C 0.000 }
gfCNCPoint1[23602] = {X 81.4951, Y 12.9779, Z -2.1667, A 0.000, B 0.000, C 0.000 }
gfCNCPoint1[23603] = {X 81.4951, Y 12.1868, Z -2.1667, A 0.000, B 0.000, C 0.000 }
gfCNCPoint1[23604] = {X 81.5776, Y 11.3388, Z -2.1667, A 0.000, B 0.000, C 0.000 }
gfCNCPoint1[23605] = {X 81.8219, Y 10.5226, Z -2.1667, A 0.000, B 0.000, C 0.000 }
gfCNCPoint1[23606] = {X 82.2190, Y 9.7689, Z -2.1667, A 0.000, B 0.000, C 0.000 }
gfCNCPoint1[23607] = {X 81.8180, Y 9.5051, Z -2.1667, A 0.000, B 0.000, C 0.000 }
gfCNCPoint1[23608] = {X 68.9232, Y 9.5051, Z -2.1667, A 0.000, B 0.000, C 0.000 }
gfCNCPoint1[23609] = {X 69.1905, Y 10.7209, Z -2.1667, A 0.000, B 0.000, C 0.000 }
gfCNCPoint1[23610] = {X 69.2995, Y 11.9611, Z -2.1667, A 0.000, B 0.000, C 0.000 }
gfCNCPoint1[23611] = {X 69.3015, Y 12.0739, Z -2.1667, A 0.000, B 0.000, C 0.000 }
gfCNCPoint1[23612] = {X 69.3021, Y 12.1868, Z -2.1667, A 0.000, B 0.000, C 0.000 }
gfCNCPoint1[23613] = {X 69.3017, Y 13.0686, Z -2.1667, A 0.000, B 0.000, C 0.000 }
gfCNCPoint1[23614] = {X 69.2132, Y 14.2874, Z -2.1667, A 0.000, B 0.000, C 0.000 }
gfCNCPoint1[23615] = {X 68.9718, Y 15.4853, Z -2.1667, A 0.000, B 0.000, C 0.000 }
gfCNCPoint1[23616] = {X 76.9172, Y 36.7523, Z -2.1667, A 0.000, B 0.000, C 0.000 }
gfCNCPoint1[23617] = {X 77.6312, Y 37.4062, Z -2.1667, A 0.000, B 0.000, C 0.000 }
gfCNCPoint1[23618] = {X 78.2763, Y 38.1281, Z -2.1667, A 0.000, B 0.000, C 0.000 }
gfCNCPoint1[23619] = {X 79.0235, Y 39.1929, Z -2.1667, A 0.000, B 0.000, C 0.000 }
gfCNCPoint1[23620] = {X 79.6213, Y 40.3482, Z -2.1667, A 0.000, B 0.000, C 0.000 }
gfCNCPoint1[23621] = {X 80.0588, Y 41.5733, Z -2.1667, A 0.000, B 0.000, C 0.000 }
gfCNCPoint1[23622] = {X 80.3280, Y 42.8459, Z -2.1667, A 0.000, B 0.000, C 0.000 }
gfCNCPoint1[23623] = {X 80.4242, Y 44.1432, Z -2.1667, A 0.000, B 0.000, C 0.000 }
gfCNCPoint1[23624] = {X 80.4245, Y 45.0000, Z -2.1667, A 0.000, B 0.000, C 0.000 }
gfCNCPoint1[23625] = {X 80.3511, Y 46.1898, Z -2.1667, A 0.000, B 0.000, C 0.000 }
gfCNCPoint1[23626] = {X 80.1320, Y 47.3615, Z -2.1667, A 0.000, B 0.000, C 0.000 }
gfCNCPoint1[23627] = {X 79.7706, Y 48.4974, Z -2.1667, A 0.000, B 0.000, C 0.000 }
gfCNCPoint1[23628] = {X 79.2722, Y 49.5803, Z -2.1667, A 0.000, B 0.000, C 0.000 }
gfCNCPoint1[23629] = {X 78.4688, Y 50.8341, Z -2.1667, A 0.000, B 0.000, C 0.000 }
gfCNCPoint1[23630] = {X 77.4826, Y 51.9498, Z -2.1667, A 0.000, B 0.000, C 0.000 }
gfCNCPoint1[23631] = {X 76.3369, Y 52.9011, Z -2.1667, A 0.000, B 0.000, C 0.000 }
gfCNCPoint1[23632] = {X 75.0589, Y 53.6653, Z -2.1667, A 0.000, B 0.000, C 0.000 }
gfCNCPoint1[23633] = {X 73.6787, Y 54.2246, Z -2.1667, A 0.000, B 0.000, C 0.000 }
gfCNCPoint1[23634] = {X 72.2292, Y 54.5655, Z -2.1667, A 0.000, B 0.000, C 0.000 }
gfCNCPoint1[23635] = {X 70.7445, Y 54.6800, Z -2.1667, A 0.000, B 0.000, C 0.000 }
gfCNCPoint1[23636] = {X 64.1851, Y 54.6800, Z -2.1667, A 0.000, B 0.000, C 0.000 }
gfCNCPoint1[23637] = {X 62.7229, Y 54.5689, Z -2.1667, A 0.000, B 0.000, C 0.000 }
gfCNCPoint1[23638] = {X 61.2943, Y 54.2383, Z -2.1667, A 0.000, B 0.000, C 0.000 }
gfCNCPoint1[23639] = {X 59.9320, Y 53.6956, Z -2.1667, A 0.000, B 0.000, C 0.000 }
gfCNCPoint1[23640] = {X 58.6673, Y 52.9534, Z -2.1667, A 0.000, B 0.000, C 0.000 }
gfCNCPoint1[23641] = {X 57.5293, Y 52.0286, Z -2.1667, A 0.000, B 0.000, C 0.000 }
gfCNCPoint1[23642] = {X 56.6337, Y 51.0563, Z -2.1667, A 0.000, B 0.000, C 0.000 }
gfCNCPoint1[23643] = {X 55.8790, Y 49.9710, Z -2.1667, A 0.000, B 0.000, C 0.000 }
gfCNCPoint1[23644] = {X 55.1243, Y 51.0563, Z -2.1667, A 0.000, B 0.000, C 0.000 }
gfCNCPoint1[23645] = {X 54.2288, Y 52.0286, Z -2.1667, A 0.000, B 0.000, C 0.000 }
gfCNCPoint1[23646] = {X 53.0907, Y 52.9534, Z -2.1667, A 0.000, B 0.000, C 0.000 }
gfCNCPoint1[23647] = {X 51.8261, Y 53.6956, Z -2.1667, A 0.000, B 0.000, C 0.000 }
gfCNCPoint1[23648] = {X 50.4638, Y 54.2383, Z -2.1667, A 0.000, B 0.000, C 0.000 }
gfCNCPoint1[23649] = {X 49.0351, Y 54.5689, Z -2.1667, A 0.000, B 0.000, C 0.000 }
gfCNCPoint1[23650] = {X 47.5729, Y 54.6800, Z -2.1667, A 0.000, B 0.000, C 0.000 }
gfCNCPoint1[23651] = {X 40.6393, Y 54.6800, Z -2.1667, A 0.000, B 0.000, C 0.000 }
gfCNCPoint1[23652] = {X 39.2448, Y 54.5790, Z -2.1667, A 0.000, B 0.000, C 0.000 }
gfCNCPoint1[23653] = {X 37.8793, Y 54.2782, Z -2.1667, A 0.000, B 0.000, C 0.000 }
gfCNCPoint1[23654] = {X 36.5715, Y 53.7838, Z -2.1667, A 0.000, B 0.000, C 0.000 }
gfCNCPoint1[23655] = {X 35.3485, Y 53.1062, Z -2.1667, A 0.000, B 0.000, C 0.000 }
gfCNCPoint1[23656] = {X 33.9156, Y 54.1338, Z -2.1667, A 0.000, B 0.000, C 0.000 }
gfCNCPoint1[23657] = {X 32.3651, Y 54.9734, Z -2.1667, A 0.000, B 0.000, C 0.000 }
gfCNCPoint1[23658] = {X 30.7214, Y 55.6118, Z -2.1667, A 0.000, B 0.000, C 0.000 }
gfCNCPoint1[23659] = {X 29.0106, Y 56.0387, Z -2.1667, A 0.000, B 0.000, C 0.000 }
gfCNCPoint1[23660] = {X 27.2597, Y 56.2475, Z -2.1667, A 0.000, B 0.000, C 0.000 }
gfCNCPoint1[23661] = {X 24.5094, Y 57.4141, Z -2.1667, A 0.000, B 0.000, C 0.000 }
gfCNCPoint1[23662] = {X 21.6764, Y 58.3621, Z -2.1667, A 0.000, B 0.000, C 0.000 }
gfCNCPoint1[23663] = {X 19.2927, Y 58.9728, Z -2.1667, A 0.000, B 0.000, C 0.000 }
gfCNCPoint1[23664] = {X 16.8694, Y 59.4003, Z -2.1667, A 0.000, B 0.000, C 0.000 }
gfCNCPoint1[23665] = {X 14.4207, Y 59.6422, Z -2.1667, A 0.000, B 0.000, C 0.000 }
gfCNCPoint1[23666] = {X 11.9606, Y 59.6970, Z -2.1667, A 0.000, B 0.000, C 0.000 }
gfCNCPoint1[23667] = {X 9.5035, Y 59.5644, Z -2.1667, A 0.000, B 0.000, C 0.000 }
gfCNCPoint1[23668] = {X 9.5035, Y 90.4949, Z -2.1667, A 0.000, B 0.000, C 0.000 }
gfCNCPoint1[23669] = {X 114.8635, Y 90.4949, Z -2.1667, A 0.000, B 0.000, C 0.000 }
gfCNCPoint1[23670] = {X 115.7479, Y 89.2990, Z -2.1667, A 0.000, B 0.000, C 0.000 }
gfCNCPoint1[23671] = {X 116.7725, Y 88.2209, Z -2.1667, A 0.000, B 0.000, C 0.000 }
gfCNCPoint1[23672] = {X 117.9219, Y 87.2768, Z -2.1667, A 0.000, B 0.000, C 0.000 }
gfCNCPoint1[23673] = {X 119.1786, Y 86.4812, Z -2.1667, A 0.000, B 0.000, C 0.000 }
gfCNCPoint1[23674] = {X 120.5235, Y 85.8460, Z -2.1667, A 0.000, B 0.000, C 0.000 }
gfCNCPoint1[23675] = {X 121.9363, Y 85.3809, Z -2.1667, A 0.000, B 0.000, C 0.000 }
gfCNCPoint1[23676] = {X 123.3956, Y 85.0930, Z -2.1667, A 0.000, B 0.000, C 0.000 }
gfCNCPoint1[23677] = {X 123.5624, Y 84.9133, Z -2.1667, A 0.000, B 0.000, C 0.000 }
gfCNCPoint1[23678] = {X 123.7274, Y 84.7320, Z -2.1667, A 0.000, B 0.000, C 0.000 }
gfCNCPoint1[23679] = {X 147.2181, Y 58.9358, Z -2.1667, A 0.000, B 0.000, C 0.000 }
gfCNCPoint1[23680] = {X 147.2180, Y 58.0000, Z -2.1667, A 0.000, B 0.000, C 0.000 }
gfCNCPoint1[23681] = {X 147.2987, Y 56.6058, Z -2.1667, A 0.000, B 0.000, C 0.000 }
gfCNCPoint1[23682] = {X 147.5398, Y 55.2303, Z -2.1667, A 0.000, B 0.000, C 0.000 }
gfCNCPoint1[23683] = {X 148.0022, Y 53.7185, Z -2.1667, A 0.000, B 0.000, C 0.000 }
gfCNCPoint1[23684] = {X 148.6580, Y 52.2800, Z -2.1667, A 0.000, B 0.000, C 0.000 }
gfCNCPoint1[23685] = {X 143.0396, Y 52.2800, Z -2.1667, A 0.000, B 0.000, C 0.000 }
gfCNCPoint1[23686] = {X 141.7807, Y 52.1703, Z -2.1667, A 0.000, B 0.000, C 0.000 }
gfCNCPoint1[23687] = {X 140.5597, Y 51.8446, Z -2.1667, A 0.000, B 0.000, C 0.000 }
gfCNCPoint1[23688] = {X 139.4134, Y 51.3126, Z -2.1667, A 0.000, B 0.000, C 0.000 }
gfCNCPoint1[23689] = {X 138.3764, Y 50.5904, Z -2.1667, A 0.000, B 0.000, C 0.000 }
gfCNCPoint1[23690] = {X 137.4799, Y 49.6998, Z -2.1667, A 0.000, B 0.000, C 0.000 }
gfCNCPoint1[23691] = {X 136.7509, Y 48.6675, Z -2.1667, A 0.000, B 0.000, C 0.000 }
gfCNCPoint1[23692] = {X 136.2114, Y 47.5248, Z -2.1667, A 0.000, B 0.000, C 0.000 }
gfCNCPoint1[23693] = {X 135.8777, Y 46.3059, Z -2.1667, A 0.000, B 0.000, C 0.000 }
gfCNCPoint1[23694] = {X 135.7598, Y 45.0477, Z -2.1667, A 0.000, B 0.000, C 0.000 }
gfCNCPoint1[23695] = {X 135.7601, Y 44.1247, Z -2.1667, A 0.000, B 0.000, C 0.000 }
gfCNCPoint1[23696] = {X 135.8408, Y 43.1249, Z -2.1667, A 0.000, B 0.000, C 0.000 }
gfCNCPoint1[23697] = {X 136.0581, Y 42.1457, Z -2.1667, A 0.000, B 0.000, C 0.000 }
gfCNCPoint1[23698] = {X 138.3597, Y 42.8258, Z -2.1667, A 0.000, B 0.000, C 0.000 }
gfCNCPoint1[23699] = {X 138.6721, Y 42.0319, Z -2.1667, A 0.000, B 0.000, C 0.000 }
gfCNCPoint1[23700] = {X 139.1179, Y 41.3046, Z -2.1667, A 0.000, B 0.000, C 0.000 }
gfCNCPoint1[23701] = {X 139.6836, Y 40.6660, Z -2.1667, A 0.000, B 0.000, C 0.000 }
gfCNCPoint1[23702] = {X 139.6836, Y 20.4366, Z -2.1667, A 0.000, B 0.000, C 0.000 }
gfCNCPoint1[23703] = {X 137.7110, Y 20.4360, Z -2.1667, A 0.000, B 0.000, C 0.000 }
gfCNCPoint1[23704] = {X 137.0004, Y 21.1818, Z -2.1667, A 0.000, B 0.000, C 0.000 }
gfCNCPoint1[23705] = {X 136.1491, Y 21.7619, Z -2.1667, A 0.000, B 0.000, C 0.000 }
gfCNCPoint1[23706] = {X 135.4282, Y 22.0767, Z -2.1667, A 0.000, B 0.000, C 0.000 }
gfCNCPoint1[23707] = {X 134.6660, Y 22.2715, Z -2.1667, A 0.000, B 0.000, C 0.000 }
gfCNCPoint1[23708] = {X 133.8824, Y 22.3414, Z -2.1667, A 0.000, B 0.000, C 0.000 }
gfCNCPoint1[23709] = {X 133.2006, Y 22.3415, Z -2.1667, A 0.000, B 0.000, C 0.000 }
gfCNCPoint1[23710] = {X 132.2486, Y 22.2478, Z -2.1667, A 0.000, B 0.000, C 0.000 }
gfCNCPoint1[23711] = {X 131.3331, Y 21.9701, Z -2.1667, A 0.000, B 0.000, C 0.000 }
gfCNCPoint1[23712] = {X 130.4895, Y 21.5191, Z -2.1667, A 0.000, B 0.000, C 0.000 }
gfCNCPoint1[23713] = {X 129.7500, Y 20.9122, Z -2.1667, A 0.000, B 0.000, C 0.000 }
gfCNCPoint1[23714] = {X 129.1431, Y 20.1727, Z -2.1667, A 0.000, B 0.000, C 0.000 }
gfCNCPoint1[23715] = {X 128.6921, Y 19.3290, Z -2.1667, A 0.000, B 0.000, C 0.000 }
gfCNCPoint1[23716] = {X 128.4144, Y 18.4136, Z -2.1667, A 0.000, B 0.000, C 0.000 }
gfCNCPoint1[23717] = {X 128.3206, Y 17.4615, Z -2.1667, A 0.000, B 0.000, C 0.000 }
gfCNCPoint1[23718] = {X 128.3206, Y 10.4835, Z -2.1667, A 0.000, B 0.000, C 0.000 }
gfCNCPoint1[23719] = {X 128.3317, Y 10.1548, Z -2.1667, A 0.000, B 0.000, C 0.000 }
gfCNCPoint1[23720] = {X 128.3649, Y 9.8276, Z -2.1667, A 0.000, B 0.000, C 0.000 }
gfCNCPoint1[23721] = {X 128.6078, Y 8.8342, Z -2.1667, A 0.000, B 0.000, C 0.000 }
gfCNCPoint1[23722] = {X 129.0524, Y 7.9132, Z -2.1667, A 0.000, B 0.000, C 0.000 }
gfCNCPoint1[23723] = {X 129.6792, Y 7.1051, Z -2.1667, A 0.000, B 0.000, C 0.000 }
gfCNCPoint1[23724] = {X 130.0256, Y 7.4374, Z -2.1667, A 0.000, B 0.000, C 0.000 }
gfCNCPoint1[23725] = {X 130.6996, Y 6.8635, Z -2.1667, A 0.000, B 0.000, C 0.000 }
gfCNCPoint1[23726] = {X 131.4748, Y 6.4361, Z -2.1667, A 0.000, B 0.000, C 0.000 }
gfCNCPoint1[23727] = {X 132.3199, Y 6.1726, Z -2.1667, A 0.000, B 0.000, C 0.000 }
gfCNCPoint1[23728] = {X 133.2007, Y 6.0835, Z -2.1667, A 0.000, B 0.000, C 0.000 }
gfCNCPoint1[23729] = {X 133.8874, Y 6.0837, Z -2.1667, A 0.000, B 0.000, C 0.000 }
gfCNCPoint1[23730] = {X 134.7191, Y 6.1718, Z -2.1667, A 0.000, B 0.000, C 0.000 }
gfCNCPoint1[23731] = {X 135.5191, Y 6.4155, Z -2.1667, A 0.000, B 0.000, C 0.000 }
gfCNCPoint1[23732] = {X 136.2585, Y 6.8063, Z -2.1667, A 0.000, B 0.000, C 0.000 }
gfCNCPoint1[23733] = {X 136.9106, Y 7.3298, Z -2.1667, A 0.000, B 0.000, C 0.000 }
gfCNCPoint1[23734] = {X 137.4519, Y 7.9674, Z -2.1667, A 0.000, B 0.000, C 0.000 }
gfCNCPoint1[23735] = {X 155.0709, Y 7.9674, Z -2.1667, A 0.000, B 0.000, C 0.000 }
gfCNCPoint1[23736] = {X 155.6186, Y 7.3235, Z -2.1667, A 0.000, B 0.000, C 0.000 }
gfCNCPoint1[23737] = {X 156.2794, Y 6.7963, Z -2.1667, A 0.000, B 0.000, C 0.000 }
gfCNCPoint1[23738] = {X 157.0288, Y 6.4052, Z -2.1667, A 0.000, B 0.000, C 0.000 }
gfCNCPoint1[23739] = {X 157.8392, Y 6.1647, Z -2.1667, A 0.000, B 0.000, C 0.000 }
gfCNCPoint1[23740] = {X 158.6806, Y 6.0835, Z -2.1667, A 0.000, B 0.000, C 0.000 }
gfCNCPoint1[23741] = {X 159.3791, Y 6.0839, Z -2.1667, A 0.000, B 0.000, C 0.000 }
gfCNCPoint1[23742] = {X 160.3488, Y 6.2050, Z -2.1667, A 0.000, B 0.000, C 0.000 }
gfCNCPoint1[23743] = {X 161.2678, Y 6.5371, Z -2.1667, A 0.000, B 0.000, C 0.000 }
gfCNCPoint1[23744] = {X 162.0908, Y 7.0639, Z -2.1667, A 0.000, B 0.000, C 0.000 }
gfCNCPoint1[23745] = {X 162.7773, Y 7.7593, Z -2.1667, A 0.000, B 0.000, C 0.000 }
gfCNCPoint1[23746] = {X 163.2934, Y 8.5891, Z -2.1667, A 0.000, B 0.000, C 0.000 }
gfCNCPoint1[23747] = {X 163.6136, Y 9.5124, Z -2.1667, A 0.000, B 0.000, C 0.000 }
gfCNCPoint1[23748] = {X 163.7221, Y 10.4835, Z -2.1667, A 0.000, B 0.000, C 0.000 }
gfCNCPoint1[23749] = {X 163.7221, Y 17.4615, Z -2.1667, A 0.000, B 0.000, C 0.000 }
gfCNCPoint1[23750] = {X 163.6118, Y 18.4406, Z -2.1667, A 0.000, B 0.000, C 0.000 }
gfCNCPoint1[23751] = {X 163.2863, Y 19.3706, Z -2.1667, A 0.000, B 0.000, C 0.000 }
gfCNCPoint1[23752] = {X 162.7621, Y 20.2049, Z -2.1667, A 0.000, B 0.000, C 0.000 }
gfCNCPoint1[23753] = {X 162.0654, Y 20.9016, Z -2.1667, A 0.000, B 0.000, C 0.000 }
gfCNCPoint1[23754] = {X 161.2312, Y 21.4258, Z -2.1667, A 0.000, B 0.000, C 0.000 }
gfCNCPoint1[23755] = {X 160.3012, Y 21.7512, Z -2.1667, A 0.000, B 0.000, C 0.000 }
gfCNCPoint1[23756] = {X 159.3221, Y 21.8615, Z -2.1667, A 0.000, B 0.000, C 0.000 }
gfCNCPoint1[23757] = {X 158.6786, Y 21.8615, Z -2.1667, A 0.000, B 0.000, C 0.000 }
gfCNCPoint1[23758] = {X 157.8333, Y 21.7761, Z -2.1667, A 0.000, B 0.000, C 0.000 }
gfCNCPoint1[23759] = {X 157.0197, Y 21.5311, Z -2.1667, A 0.000, B 0.000, C 0.000 }
gfCNCPoint1[23760] = {X 156.2677, Y 21.1356, Z -2.1667, A 0.000, B 0.000, C 0.000 }
gfCNCPoint1[23761] = {X 155.6049, Y 20.6041, Z -2.1667, A 0.000, B 0.000, C 0.000 }
gfCNCPoint1[23762] = {X 155.0554, Y 19.9560, Z -2.1667, A 0.000, B 0.000, C 0.000 }
gfCNCPoint1[23763] = {X 152.3557, Y 19.9573, Z -2.1667, A 0.000, B 0.000, C 0.000 }
gfCNCPoint1[23764] = {X 152.3541, Y 40.8428, Z -2.1667, A 0.000, B 0.000, C 0.000 }
gfCNCPoint1[23765] = {X 152.8076, Y 41.3317, Z -2.1667, A 0.000, B 0.000, C 0.000 }
gfCNCPoint1[23766] = {X 152.8991, Y 41.4411, Z -2.1667, A 0.000, B 0.000, C 0.000 }
gfCNCPoint1[23767] = {X 153.4334, Y 42.2815, Z -2.1667, A 0.000, B 0.000, C 0.000 }
gfCNCPoint1[23768] = {X 153.7670, Y 43.2198, Z -2.1667, A 0.000, B 0.000, C 0.000 }
gfCNCPoint1[23769] = {X 153.8831, Y 44.2089, Z -2.1667, A 0.000, B 0.000, C 0.000 }
gfCNCPoint1[23770] = {X 153.8829, Y 45.0423, Z -2.1667, A 0.000, B 0.000, C 0.000 }
gfCNCPoint1[23771] = {X 153.7646, Y 46.0144, Z -2.1667, A 0.000, B 0.000, C 0.000 }
gfCNCPoint1[23772] = {X 153.4342, Y 46.9363, Z -2.1667, A 0.000, B 0.000, C 0.000 }
gfCNCPoint1[23773] = {X 152.9080, Y 47.7622, Z -2.1667, A 0.000, B 0.000, C 0.000 }
gfCNCPoint1[23774] = {X 152.2123, Y 48.4513, Z -2.1667, A 0.000, B 0.000, C 0.000 }
gfCNCPoint1[23775] = {X 151.3813, Y 48.9695, Z -2.1667, A 0.000, B 0.000, C 0.000 }
gfCNCPoint1[23776] = {X 150.4563, Y 49.2910, Z -2.1667, A 0.000, B 0.000, C 0.000 }
gfCNCPoint1[23777] = {X 149.4831, Y 49.4000, Z -2.1667, A 0.000, B 0.000, C 0.000 }
gfCNCPoint1[23778] = {X 143.0396, Y 49.4000, Z -2.1667, A 0.000, B 0.000, C 0.000 }
gfCNCPoint1[23779] = {X 142.0605, Y 49.2897, Z -2.1667, A 0.000, B 0.000, C 0.000 }
gfCNCPoint1[23780] = {X 141.1305, Y 48.9643, Z -2.1667, A 0.000, B 0.000, C 0.000 }
gfCNCPoint1[23781] = {X 140.2963, Y 48.4400, Z -2.1667, A 0.000, B 0.000, C 0.000 }
gfCNCPoint1[23782] = {X 139.5996, Y 47.7433, Z -2.1667, A 0.000, B 0.000, C 0.000 }
gfCNCPoint1[23783] = {X 139.0754, Y 46.9091, Z -2.1667, A 0.000, B 0.000, C 0.000 }
gfCNCPoint1[23784] = {X 138.7499, Y 45.9791, Z -2.1667, A 0.000, B 0.000, C 0.000 }
gfCNCPoint1[23785] = {X 138.6396, Y 45.0000, Z -2.1667, A 0.000, B 0.000, C 0.000 }
gfCNCPoint1[23786] = {X 138.6400, Y 44.1483, Z -2.1667, A 0.000, B 0.000, C 0.000 }
gfCNCPoint1[23787] = {X 138.7505, Y 43.2275, Z -2.1667, A 0.000, B 0.000, C 0.000 }
gfCNCPoint1[23788] = {X 139.0514, Y 42.3503, Z -2.1667, A 0.000, B 0.000, C 0.000 }
gfCNCPoint1[23789] = {X 139.5295, Y 41.5556, Z -2.1667, A 0.000, B 0.000, C 0.000 }
gfCNCPoint1[23790] = {X 140.1636, Y 40.8789, Z -2.1667, A 0.000, B 0.000, C 0.000 }
gfCNCPoint1[23791] = {X 140.1636, Y 19.9567, Z -2.1667, A 0.000, B 0.000, C 0.000 }
gfCNCPoint1[23792] = {X 137.4670, Y 19.9559, Z -2.1667, A 0.000, B 0.000, C 0.000 }
gfCNCPoint1[23793] = {X 136.9193, Y 20.6067, Z -2.1667, A 0.000, B 0.000, C 0.000 }
gfCNCPoint1[23794] = {X 136.2566, Y 21.1400, Z -2.1667, A 0.000, B 0.000, C 0.000 }
gfCNCPoint1[23795] = {X 135.5037, Y 21.5358, Z -2.1667, A 0.000, B 0.000, C 0.000 }
gfCNCPoint1[23796] = {X 134.6887, Y 21.7794, Z -2.1667, A 0.000, B 0.000, C 0.000 }
gfCNCPoint1[23797] = {X 133.8421, Y 21.8615, Z -2.1667, A 0.000, B 0.000, C 0.000 }
gfCNCPoint1[23798] = {X 133.2006, Y 21.8615, Z -2.1667, A 0.000, B 0.000, C 0.000 }
gfCNCPoint1[23799] = {X 132.2215, Y 21.7512, Z -2.1667, A 0.000, B 0.000, C 0.000 }
gfCNCPoint1[23800] = {X 131.2916, Y 21.4258, Z -2.1667, A 0.000, B 0.000, C 0.000 }
gfCNCPoint1[23801] = {X 130.4573, Y 20.9016, Z -2.1667, A 0.000, B 0.000, C 0.000 }
gfCNCPoint1[23802] = {X 129.7606, Y 20.2049, Z -2.1667, A 0.000, B 0.000, C 0.000 }
gfCNCPoint1[23803] = {X 129.2364, Y 19.3706, Z -2.1667, A 0.000, B 0.000, C 0.000 }
gfCNCPoint1[23804] = {X 128.9110, Y 18.4406, Z -2.1667, A 0.000, B 0.000, C 0.000 }
gfCNCPoint1[23805] = {X 128.8006, Y 17.4615, Z -2.1667, A 0.000, B 0.000, C 0.000 }
gfCNCPoint1[23806] = {X 128.8006, Y 10.4835, Z -2.1667, A 0.000, B 0.000, C 0.000 }
gfCNCPoint1[23807] = {X 128.8808, Y 9.6475, Z -2.1667, A 0.000, B 0.000, C 0.000 }
gfCNCPoint1[23808] = {X 129.1183, Y 8.8419, Z -2.1667, A 0.000, B 0.000, C 0.000 }
gfCNCPoint1[23809] = {X 129.5046, Y 8.0962, Z -2.1667, A 0.000, B 0.000, C 0.000 }
gfCNCPoint1[23810] = {X 130.0256, Y 7.4374, Z -2.1667, A 0.000, B 0.000, C 0.000 }
gfCNCPoint1[23811] = {X 129.6792, Y 7.1051, Z -2.1667, A 0.000, B 0.000, C 0.000 }
gfCNCPoint1[23812] = {X 102.4337, Y 7.1051, Z -2.1667, A 0.000, B 0.000, C 0.000 }
gfCNCPoint1[23813] = {X 102.4337, Y 11.9051, Z -2.1667, A 0.000, B 0.000, C 0.000 }
gfCNCPoint1[23814] = {X 101.3242, Y 11.9051, Z -2.1667, A 0.000, B 0.000, C 0.000 }
gfCNCPoint1[23815] = {X 101.3283, Y 12.0459, Z -2.1667, A 0.000, B 0.000, C 0.000 }
gfCNCPoint1[23816] = {X 101.3297, Y 12.1868, Z -2.1667, A 0.000, B 0.000, C 0.000 }
gfCNCPoint1[23817] = {X 101.3293, Y 13.0462, Z -2.1667, A 0.000, B 0.000, C 0.000 }
gfCNCPoint1[23818] = {X 101.2273, Y 14.1943, Z -2.1667, A 0.000, B 0.000, C 0.000 }
gfCNCPoint1[23819] = {X 100.9454, Y 15.3120, Z -2.1667, A 0.000, B 0.000, C 0.000 }
gfCNCPoint1[23820] = {X 101.0386, Y 15.5442, Z -2.1667, A 0.000, B 0.000, C 0.000 }
gfCNCPoint1[23821] = {X 101.8684, Y 17.6011, Z -2.1667, A 0.000, B 0.000, C 0.000 }
gfCNCPoint1[23822] = {X 102.8006, Y 15.2764, Z -2.1667, A 0.000, B 0.000, C 0.000 }
gfCNCPoint1[23823] = {X 102.5274, Y 14.1754, Z -2.1667, A 0.000, B 0.000, C 0.000 }
gfCNCPoint1[23824] = {X 102.4286, Y 13.0453, Z -2.1667, A 0.000, B 0.000, C 0.000 }
gfCNCPoint1[23825] = {X 102.4283, Y 12.1868, Z -2.1667, A 0.000, B 0.000, C 0.000 }
gfCNCPoint1[23826] = {X 102.4296, Y 12.0459, Z -2.1667, A 0.000, B 0.000, C 0.000 }
gfCNCPoint1[23827] = {X 102.4337, Y 11.9051, Z -2.1667, A 0.000, B 0.000, C 0.000 }
gfCNCPoint1[23828] = {X 102.4337, Y 9.5051, Z -2.1667, A 0.000, B 0.000, C 0.000 }
gfCNCPoint1[23829] = {X 98.1268, Y 9.5051, Z -2.1667, A 0.000, B 0.000, C 0.000 }
gfCNCPoint1[23830] = {X 98.5430, Y 10.2830, Z -2.1667, A 0.000, B 0.000, C 0.000 }
gfCNCPoint1[23831] = {X 98.8123, Y 11.1231, Z -2.1667, A 0.000, B 0.000, C 0.000 }
gfCNCPoint1[23832] = {X 98.9260, Y 11.9980, Z -2.1667, A 0.000, B 0.000, C 0.000 }
gfCNCPoint1[23833] = {X 98.9288, Y 12.0924, Z -2.1667, A 0.000, B 0.000, C 0.000 }
gfCNCPoint1[23834] = {X 98.9297, Y 12.1868, Z -2.1667, A 0.000, B 0.000, C 0.000 }
gfCNCPoint1[23835] = {X 98.9294, Y 13.0237, Z -2.1667, A 0.000, B 0.000, C 0.000 }
gfCNCPoint1[23836] = {X 98.8589, Y 13.8061, Z -2.1667, A 0.000, B 0.000, C 0.000 }
gfCNCPoint1[23837] = {X 98.6637, Y 14.5671, Z -2.1667, A 0.000, B 0.000, C 0.000 }
gfCNCPoint1[23838] = {X 98.3489, Y 15.2869, Z -2.1667, A 0.000, B 0.000, C 0.000 }
gfCNCPoint1[23839] = {X 98.8122, Y 16.4404, Z -2.1667, A 0.000, B 0.000, C 0.000 }
gfCNCPoint1[23840] = {X 101.8752, Y 24.0328, Z -2.1667, A 0.000, B 0.000, C 0.000 }
gfCNCPoint1[23841] = {X 105.3937, Y 15.2581, Z -2.1667, A 0.000, B 0.000, C 0.000 }
gfCNCPoint1[23842] = {X 105.0871, Y 14.5463, Z -2.1667, A 0.000, B 0.000, C 0.000 }
gfCNCPoint1[23843] = {X 104.8971, Y 13.7950, Z -2.1667, A 0.000, B 0.000, C 0.000 }
gfCNCPoint1[23844] = {X 104.8285, Y 13.0231, Z -2.1667, A 0.000, B 0.000, C 0.000 }
gfCNCPoint1[23845] = {X 104.8283, Y 12.1868, Z -2.1667, A 0.000, B 0.000, C 0.000 }
gfCNCPoint1[23846] = {X 104.8292, Y 12.0924, Z -2.1667, A 0.000, B 0.000, C 0.000 }
gfCNCPoint1[23847] = {X 104.8319, Y 11.9980, Z -2.1667, A 0.000, B 0.000, C 0.000 }
gfCNCPoint1[23848] = {X 104.9456, Y 11.1231, Z -2.1667, A 0.000, B 0.000, C 0.000 }
gfCNCPoint1[23849] = {X 105.2150, Y 10.2830, Z -2.1667, A 0.000, B 0.000, C 0.000 }
gfCNCPoint1[23850] = {X 105.6312, Y 9.5051, Z -2.1667, A 0.000, B 0.000, C 0.000 }
gfCNCPoint1[23851] = {X 102.4337, Y 9.5051, Z -2.1667, A 0.000, B 0.000, C 0.000 }
gfCNCPoint1[23852] = {X 102.4337, Y 7.1051, Z -2.1667, A 0.000, B 0.000, C 0.000 }
gfCNCPoint1[23853] = {X 64.8350, Y 7.1051, Z -2.1667, A 0.000, B 0.000, C 0.000 }
gfCNCPoint1[23854] = {X 65.5947, Y 8.0242, Z -2.1667, A 0.000, B 0.000, C 0.000 }
gfCNCPoint1[23855] = {X 66.1941, Y 9.0551, Z -2.1667, A 0.000, B 0.000, C 0.000 }
gfCNCPoint1[23856] = {X 66.6172, Y 10.1700, Z -2.1667, A 0.000, B 0.000, C 0.000 }
gfCNCPoint1[23857] = {X 66.8305, Y 11.1684, Z -2.1667, A 0.000, B 0.000, C 0.000 }
gfCNCPoint1[23858] = {X 66.9021, Y 12.1868, Z -2.1667, A 0.000, B 0.000, C 0.000 }
gfCNCPoint1[23859] = {X 66.9018, Y 13.0462, Z -2.1667, A 0.000, B 0.000, C 0.000 }
gfCNCPoint1[23860] = {X 66.7778, Y 14.3179, Z -2.1667, A 0.000, B 0.000, C 0.000 }
gfCNCPoint1[23861] = {X 66.4333, Y 15.5483, Z -2.1667, A 0.000, B 0.000, C 0.000 }
gfCNCPoint1[23862] = {X 74.9105, Y 38.2387, Z -2.1667, A 0.000, B 0.000, C 0.000 }
gfCNCPoint1[23863] = {X 75.8031, Y 38.9734, Z -2.1667, A 0.000, B 0.000, C 0.000 }
gfCNCPoint1[23864] = {X 76.5681, Y 39.8403, Z -2.1667, A 0.000, B 0.000, C 0.000 }
gfCNCPoint1[23865] = {X 77.1862, Y 40.8172, Z -2.1667, A 0.000, B 0.000, C 0.000 }
gfCNCPoint1[23866] = {X 77.6419, Y 41.8798, Z -2.1667, A 0.000, B 0.000, C 0.000 }
gfCNCPoint1[23867] = {X 77.9236, Y 43.0010, Z -2.1667, A 0.000, B 0.000, C 0.000 }
gfCNCPoint1[23868] = {X 78.0243, Y 44.1527, Z -2.1667, A 0.000, B 0.000, C 0.000 }
gfCNCPoint1[23869] = {X 78.0245, Y 45.0000, Z -2.1667, A 0.000, B 0.000, C 0.000 }
gfCNCPoint1[23870] = {X 77.9139, Y 46.2642, Z -2.1667, A 0.000, B 0.000, C 0.000 }
gfCNCPoint1[23871] = {X 77.5854, Y 47.4899, Z -2.1667, A 0.000, B 0.000, C 0.000 }
gfCNCPoint1[23872] = {X 77.0491, Y 48.6400, Z -2.1667, A 0.000, B 0.000, C 0.000 }
gfCNCPoint1[23873] = {X 76.3213, Y 49.6795, Z -2.1667, A 0.000, B 0.000, C 0.000 }
gfCNCPoint1[23874] = {X 75.4240, Y 50.5768, Z -2.1667, A 0.000, B 0.000, C 0.000 }
gfCNCPoint1[23875] = {X 74.3845, Y 51.3047, Z -2.1667, A 0.000, B 0.000, C 0.000 }
gfCNCPoint1[23876] = {X 73.2344, Y 51.8410, Z -2.1667, A 0.000, B 0.000, C 0.000 }
gfCNCPoint1[23877] = {X 72.0086, Y 52.1694, Z -2.1667, A 0.000, B 0.000, C 0.000 }
gfCNCPoint1[23878] = {X 70.7445, Y 52.2800, Z -2.1667, A 0.000, B 0.000, C 0.000 }
gfCNCPoint1[23879] = {X 64.1851, Y 52.2800, Z -2.1667, A 0.000, B 0.000, C 0.000 }
gfCNCPoint1[23880] = {X 62.9397, Y 52.1727, Z -2.1667, A 0.000, B 0.000, C 0.000 }
gfCNCPoint1[23881] = {X 61.7311, Y 51.8539, Z -2.1667, A 0.000, B 0.000, C 0.000 }
gfCNCPoint1[23882] = {X 60.5947, Y 51.3330, Z -2.1667, A 0.000, B 0.000, C 0.000 }
gfCNCPoint1[23883] = {X 59.5643, Y 50.6255, Z -2.1667, A 0.000, B 0.000, C 0.000 }
gfCNCPoint1[23884] = {X 58.6700, Y 49.7521, Z -2.1667, A 0.000, B 0.000, C 0.000 }
gfCNCPoint1[23885] = {X 57.9384, Y 48.7385, Z -2.1667, A 0.000, B 0.000, C 0.000 }
gfCNCPoint1[23886] = {X 57.3706, Y 47.5614, Z -2.1667, A 0.000, B 0.000, C 0.000 }
gfCNCPoint1[23887] = {X 57.0224, Y 46.3017, Z -2.1667, A 0.000, B 0.000, C 0.000 }
gfCNCPoint1[23888] = {X 56.9051, Y 45.0000, Z -2.1667, A 0.000, B 0.000, C 0.000 }
gfCNCPoint1[23889] = {X 56.9052, Y 44.1969, Z -2.1667, A 0.000, B 0.000, C 0.000 }
gfCNCPoint1[23890] = {X 56.9289, Y 43.6212, Z -2.1667, A 0.000, B 0.000, C 0.000 }
gfCNCPoint1[23891] = {X 56.9981, Y 43.0492, Z -2.1667, A 0.000, B 0.000, C 0.000 }
gfCNCPoint1[23892] = {X 54.7600, Y 43.0492, Z -2.1667, A 0.000, B 0.000, C 0.000 }
gfCNCPoint1[23893] = {X 54.8275, Y 43.6012, Z -2.1667, A 0.000, B 0.000, C 0.000 }
gfCNCPoint1[23894] = {X 54.8528, Y 44.1567, Z -2.1667, A 0.000, B 0.000, C 0.000 }
gfCNCPoint1[23895] = {X 54.8529, Y 45.0000, Z -2.1667, A 0.000, B 0.000, C 0.000 }
gfCNCPoint1[23896] = {X 54.7356, Y 46.3017, Z -2.1667, A 0.000, B 0.000, C 0.000 }
gfCNCPoint1[23897] = {X 54.3875, Y 47.5614, Z -2.1667, A 0.000, B 0.000, C 0.000 }
gfCNCPoint1[23898] = {X 53.8197, Y 48.7385, Z -2.1667, A 0.000, B 0.000, C 0.000 }
gfCNCPoint1[23899] = {X 53.0880, Y 49.7521, Z -2.1667, A 0.000, B 0.000, C 0.000 }
gfCNCPoint1[23900] = {X 52.1938, Y 50.6255, Z -2.1667, A 0.000, B 0.000, C 0.000 }
gfCNCPoint1[23901] = {X 51.1633, Y 51.3330, Z -2.1667, A 0.000, B 0.000, C 0.000 }
gfCNCPoint1[23902] = {X 50.0270, Y 51.8539, Z -2.1667, A 0.000, B 0.000, C 0.000 }
gfCNCPoint1[23903] = {X 48.8183, Y 52.1727, Z -2.1667, A 0.000, B 0.000, C 0.000 }
gfCNCPoint1[23904] = {X 47.5729, Y 52.2800, Z -2.1667, A 0.000, B 0.000, C 0.000 }
gfCNCPoint1[23905] = {X 40.6393, Y 52.2800, Z -2.1667, A 0.000, B 0.000, C 0.000 }
gfCNCPoint1[23906] = {X 39.4476, Y 52.1818, Z -2.1667, A 0.000, B 0.000, C 0.000 }
gfCNCPoint1[23907] = {X 38.2881, Y 51.8899, Z -2.1667, A 0.000, B 0.000, C 0.000 }
gfCNCPoint1[23908] = {X 37.1919, Y 51.4120, Z -2.1667, A 0.000, B 0.000, C 0.000 }
gfCNCPoint1[23909] = {X 36.1888, Y 50.7612, Z -2.1667, A 0.000, B 0.000, C 0.000 }
gfCNCPoint1[23910] = {X 35.3058, Y 49.9550, Z -2.1667, A 0.000, B 0.000, C 0.000 }
gfCNCPoint1[23911] = {X 34.8234, Y 50.4196, Z -2.1667, A 0.000, B 0.000, C 0.000 }
gfCNCPoint1[23912] = {X 34.3150, Y 50.8555, Z -2.1667, A 0.000, B 0.000, C 0.000 }
gfCNCPoint1[23913] = {X 33.7712, Y 51.2951, Z -2.1667, A 0.000, B 0.000, C 0.000 }
gfCNCPoint1[23914] = {X 32.5136, Y 52.1787, Z -2.1667, A 0.000, B 0.000, C 0.000 }
gfCNCPoint1[23915] = {X 31.1504, Y 52.8885, Z -2.1667, A 0.000, B 0.000, C 0.000 }
gfCNCPoint1[23916] = {X 29.7054, Y 53.4121, Z -2.1667, A 0.000, B 0.000, C 0.000 }
gfCNCPoint1[23917] = {X 28.2039, Y 53.7404, Z -2.1667, A 0.000, B 0.000, C 0.000 }
gfCNCPoint1[23918] = {X 26.6722, Y 53.8676, Z -2.1667, A 0.000, B 0.000, C 0.000 }
gfCNCPoint1[23919] = {X 24.8234, Y 54.7053, Z -2.1667, A 0.000, B 0.000, C 0.000 }
gfCNCPoint1[23920] = {X 22.9302, Y 55.4368, Z -2.1667, A 0.000, B 0.000, C 0.000 }
gfCNCPoint1[23921] = {X 20.9985, Y 56.0598, Z -2.1667, A 0.000, B 0.000, C 0.000 }
gfCNCPoint1[23922] = {X 18.7908, Y 56.6259, Z -2.1667, A 0.000, B 0.000, C 0.000 }
gfCNCPoint1[23923] = {X 16.5464, Y 57.0222, Z -2.1667, A 0.000, B 0.000, C 0.000 }
gfCNCPoint1[23924] = {X 14.2783, Y 57.2464, Z -2.1667, A 0.000, B 0.000, C 0.000 }
gfCNCPoint1[23925] = {X 11.9998, Y 57.2973, Z -2.1667, A 0.000, B 0.000, C 0.000 }
gfCNCPoint1[23926] = {X 9.7240, Y 57.1746, Z -2.1667, A 0.000, B 0.000, C 0.000 }
gfCNCPoint1[23927] = {X 8.4098, Y 57.0240, Z -2.1667, A 0.000, B 0.000, C 0.000 }
gfCNCPoint1[23928] = {X 7.1035, Y 56.8154, Z -2.1667, A 0.000, B 0.000, C 0.000 }
gfCNCPoint1[23929] = {X 7.1035, Y 92.8949, Z -2.1667, A 0.000, B 0.000, C 0.000 }
gfCNCPoint1[23930] = {X 116.2647, Y 92.8949, Z -2.1667, A 0.000, B 0.000, C 0.000 }
gfCNCPoint1[23931] = {X 116.9728, Y 91.6561, Z -2.1667, A 0.000, B 0.000, C 0.000 }
gfCNCPoint1[23932] = {X 117.8552, Y 90.5349, Z -2.1667, A 0.000, B 0.000, C 0.000 }
gfCNCPoint1[23933] = {X 118.8929, Y 89.5555, Z -2.1667, A 0.000, B 0.000, C 0.000 }
gfCNCPoint1[23934] = {X 120.0633, Y 88.7394, Z -2.1667, A 0.000, B 0.000, C 0.000 }
gfCNCPoint1[23935] = {X 121.3410, Y 88.1041, Z -2.1667, A 0.000, B 0.000, C 0.000 }
gfCNCPoint1[23936] = {X 122.6982, Y 87.6636, Z -2.1667, A 0.000, B 0.000, C 0.000 }
gfCNCPoint1[23937] = {X 124.1053, Y 87.4274, Z -2.1667, A 0.000, B 0.000, C 0.000 }
gfCNCPoint1[23938] = {X 124.5364, Y 87.3624, Z -2.1667, A 0.000, B 0.000, C 0.000 }
gfCNCPoint1[23939] = {X 125.0284, Y 86.8593, Z -2.1667, A 0.000, B 0.000, C 0.000 }
gfCNCPoint1[23940] = {X 125.5064, Y 86.3429, Z -2.1667, A 0.000, B 0.000, C 0.000 }
gfCNCPoint1[23941] = {X 149.6586, Y 59.8204, Z -2.1667, A 0.000, B 0.000, C 0.000 }
gfCNCPoint1[23942] = {X 149.6295, Y 59.4071, Z -2.1667, A 0.000, B 0.000, C 0.000 }
gfCNCPoint1[23943] = {X 149.6181, Y 58.9930, Z -2.1667, A 0.000, B 0.000, C 0.000 }
gfCNCPoint1[23944] = {X 149.6180, Y 58.0000, Z -2.1667, A 0.000, B 0.000, C 0.000 }
gfCNCPoint1[23945] = {X 149.6915, Y 56.8093, Z -2.1667, A 0.000, B 0.000, C 0.000 }
gfCNCPoint1[23946] = {X 149.9109, Y 55.6367, Z -2.1667, A 0.000, B 0.000, C 0.000 }
gfCNCPoint1[23947] = {X 150.2729, Y 54.5000, Z -2.1667, A 0.000, B 0.000, C 0.000 }
gfCNCPoint1[23948] = {X 150.7719, Y 53.4164, Z -2.1667, A 0.000, B 0.000, C 0.000 }
gfCNCPoint1[23949] = {X 151.5117, Y 52.2488, Z -2.1667, A 0.000, B 0.000, C 0.000 }
gfCNCPoint1[23950] = {X 152.4103, Y 51.1984, Z -2.1667, A 0.000, B 0.000, C 0.000 }
gfCNCPoint1[23951] = {X 153.4493, Y 50.2867, Z -2.1667, A 0.000, B 0.000, C 0.000 }
gfCNCPoint1[23952] = {X 154.6075, Y 49.5323, Z -2.1667, A 0.000, B 0.000, C 0.000 }
gfCNCPoint1[23953] = {X 155.8614, Y 48.9505, Z -2.1667, A 0.000, B 0.000, C 0.000 }
gfCNCPoint1[23954] = {X 157.1854, Y 48.5533, Z -2.1667, A 0.000, B 0.000, C 0.000 }
gfCNCPoint1[23955] = {X 158.2353, Y 48.3785, Z -2.1667, A 0.000, B 0.000, C 0.000 }
gfCNCPoint1[23956] = {X 159.2980, Y 48.3200, Z -2.1667, A 0.000, B 0.000, C 0.000 }
gfCNCPoint1[23957] = {X 176.3116, Y 48.3200, Z -2.1667, A 0.000, B 0.000, C 0.000 }
gfCNCPoint1[23958] = {X 175.1966, Y 47.6605, Z -2.1667, A 0.000, B 0.000, C 0.000 }
gfCNCPoint1[23959] = {X 174.1332, Y 46.9208, Z -2.1667, A 0.000, B 0.000, C 0.000 }
gfCNCPoint1[23960] = {X 172.7676, Y 45.7584, Z -2.1667, A 0.000, B 0.000, C 0.000 }
gfCNCPoint1[23961] = {X 171.5644, Y 44.4288, Z -2.1667, A 0.000, B 0.000, C 0.000 }
gfCNCPoint1[23962] = {X 170.6264, Y 43.0901, Z -2.1667, A 0.000, B 0.000, C 0.000 }
gfCNCPoint1[23963] = {X 169.8534, Y 41.6499, Z -2.1667, A 0.000, B 0.000, C 0.000 }
gfCNCPoint1[23964] = {X 169.2561, Y 40.1283, Z -2.1667, A 0.000, B 0.000, C 0.000 }
gfCNCPoint1[23965] = {X 168.8430, Y 38.5468, Z -2.1667, A 0.000, B 0.000, C 0.000 }
gfCNCPoint1[23966] = {X 168.6199, Y 36.9276, Z -2.1667, A 0.000, B 0.000, C 0.000 }
gfCNCPoint1[23967] = {X 168.5335, Y 35.0261, Z -2.1667, A 0.000, B 0.000, C 0.000 }
gfCNCPoint1[23968] = {X 168.6856, Y 33.1288, Z -2.1667, A 0.000, B 0.000, C 0.000 }
gfCNCPoint1[23969] = {X 169.0737, Y 31.2653, Z -2.1667, A 0.000, B 0.000, C 0.000 }
gfCNCPoint1[23970] = {X 169.6918, Y 29.4650, Z -2.1667, A 0.000, B 0.000, C 0.000 }
gfCNCPoint1[23971] = {X 170.2640, Y 28.2683, Z -2.1667, A 0.000, B 0.000, C 0.000 }
gfCNCPoint1[23972] = {X 170.9710, Y 27.1459, Z -2.1667, A 0.000, B 0.000, C 0.000 }
gfCNCPoint1[23973] = {X 171.8034, Y 26.1131, Z -2.1667, A 0.000, B 0.000, C 0.000 }
gfCNCPoint1[23974] = {X 172.7499, Y 25.1837, Z -2.1667, A 0.000, B 0.000, C 0.000 }
gfCNCPoint1[23975] = {X 173.7978, Y 24.3703, Z -2.1667, A 0.000, B 0.000, C 0.000 }
gfCNCPoint1[23976] = {X 173.0273, Y 23.7520, Z -2.1667, A 0.000, B 0.000, C 0.000 }
gfCNCPoint1[23977] = {X 172.3972, Y 22.9913, Z -2.1667, A 0.000, B 0.000, C 0.000 }
gfCNCPoint1[23978] = {X 171.9332, Y 22.1192, Z -2.1667, A 0.000, B 0.000, C 0.000 }
gfCNCPoint1[23979] = {X 169.3220, Y 15.7237, Z -2.1667, A 0.000, B 0.000, C 0.000 }
gfCNCPoint1[23980] = {X 169.1088, Y 15.0753, Z -2.1667, A 0.000, B 0.000, C 0.000 }
gfCNCPoint1[23981] = {X 168.9882, Y 14.4035, Z -2.1667, A 0.000, B 0.000, C 0.000 }
gfCNCPoint1[23982] = {X 168.9599, Y 13.8791, Z -2.1667, A 0.000, B 0.000, C 0.000 }
gfCNCPoint1[23983] = {X 168.9882, Y 13.3548, Z -2.1667, A 0.000, B 0.000, C 0.000 }
gfCNCPoint1[23984] = {X 169.1590, Y 12.4995, Z -2.1667, A 0.000, B 0.000, C 0.000 }
gfCNCPoint1[23985] = {X 169.4794, Y 11.6883, Z -2.1667, A 0.000, B 0.000, C 0.000 }
gfCNCPoint1[23986] = {X 169.9390, Y 10.9471, Z -2.1667, A 0.000, B 0.000, C 0.000 }
gfCNCPoint1[23987] = {X 170.6134, Y 10.2180, Z -2.1667, A 0.000, B 0.000, C 0.000 }
gfCNCPoint1[23988] = {X 171.4215, Y 9.6405, Z -2.1667, A 0.000, B 0.000, C 0.000 }
gfCNCPoint1[23989] = {X 172.0576, Y 9.2779, Z -2.1667, A 0.000, B 0.000, C 0.000 }
gfCNCPoint1[23990] = {X 172.9937, Y 8.8768, Z -2.1667, A 0.000, B 0.000, C 0.000 }
gfCNCPoint1[23991] = {X 173.9927, Y 8.6787, Z -2.1667, A 0.000, B 0.000, C 0.000 }
gfCNCPoint1[23992] = {X 175.0111, Y 8.6923, Z -2.1667, A 0.000, B 0.000, C 0.000 }
gfCNCPoint1[23993] = {X 176.0045, Y 8.9170, Z -2.1667, A 0.000, B 0.000, C 0.000 }
gfCNCPoint1[23994] = {X 177.7790, Y 8.1690, Z -2.1667, A 0.000, B 0.000, C 0.000 }
gfCNCPoint1[23995] = {X 179.6072, Y 7.5638, Z -2.1667, A 0.000, B 0.000, C 0.000 }
gfCNCPoint1[23996] = {X 181.4776, Y 7.1051, Z -2.1667, A 0.000, B 0.000, C 0.000 }
gfCNCPoint1[23997] = {X 168.0205, Y 7.1051, Z -2.1667, A 0.000, B 0.000, C 0.000 }
gfCNCPoint1[23998] = {X 168.0205, Y 4.7051, Z -2.1667, A 0.000, B 0.000, C 0.000 }
gfCNCPoint1[23999] = {X 155.1590, Y 4.7051, Z -2.1667, A 0.000, B 0.000, C 0.000 }
gfCNCPoint1[24000] = {X 155.1590, Y 7.1051, Z -2.1667, A 0.000, B 0.000, C 0.000 }
gfCNCPoint1[24001] = {X 137.3638, Y 7.1051, Z -2.1667, A 0.000, B 0.000, C 0.000 }
gfCNCPoint1[24002] = {X 137.5340, Y 7.2919, Z -2.1667, A 0.000, B 0.000, C 0.000 }
gfCNCPoint1[24003] = {X 137.6942, Y 7.4874, Z -2.1667, A 0.000, B 0.000, C 0.000 }
gfCNCPoint1[24004] = {X 154.8285, Y 7.4874, Z -2.1667, A 0.000, B 0.000, C 0.000 }
gfCNCPoint1[24005] = {X 154.9888, Y 7.2919, Z -2.1667, A 0.000, B 0.000, C 0.000 }
gfCNCPoint1[24006] = {X 155.1590, Y 7.1051, Z -2.1667, A 0.000, B 0.000, C 0.000 }
gfCNCPoint1[24007] = {X 155.1590, Y 4.7051, Z -2.1667, A 0.000, B 0.000, C 0.000 }
gfCNCPoint1[24008] = {X 23.8340, Y 4.7051, Z -2.1667, A 0.000, B 0.000, C 0.000 }
